Yaskawa INFORM job: test_long_tjr5.JBI

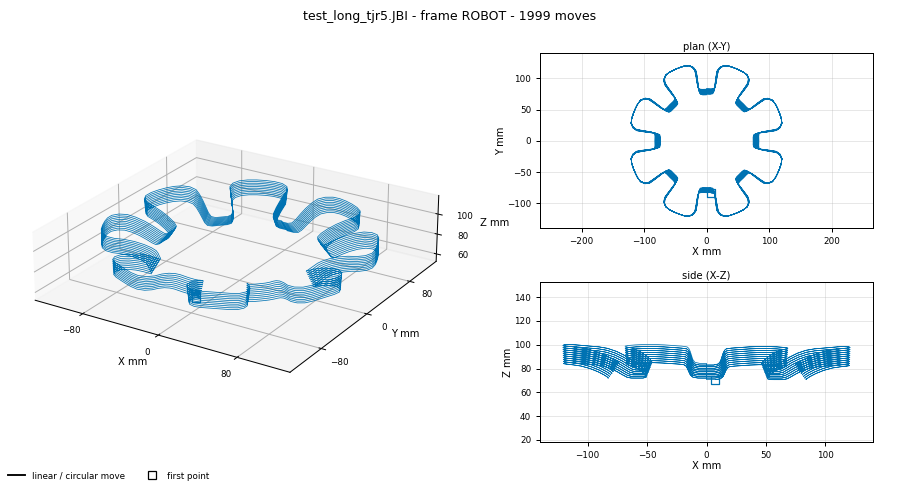
[picture p0: tool path of test_long_tjr5.JBI in frame ROBOT, 1999 of 2000 moves have a stored position in this frame; points joined in program order, loops and branches not executed]
version: 0
/JOB
//NAME test_long
//POS
///NPOS 48,0,0,2,0,0
///TOOL 1
///POSTYPE ROBOT
///RECTAN
///RCONF 1,0,0,0,0,0,0,0,0,0,0,0,0,0,0,0,0,0,0,0,0,0,0,0
C00000=3.480,-83.770,70.680,-0.0300,0.6200,0.7800
C00001=7.410,-83.590,70.710,0.0200,0.6100,0.7900
C00002=11.710,-84.200,71.430,0.2600,0.4000,0.8800
C00003=13.880,-86.990,73.260,0.0400,0.0100,1.0000
C00004=15.150,-91.900,75.810,-0.0600,-0.0100,1.0000
C00005=16.340,-98.510,78.470,-0.1100,-0.0200,0.9900
C00006=17.620,-105.970,80.520,-0.1300,-0.0300,0.9900
C00007=19.220,-112.910,81.540,-0.1300,-0.0600,0.9900
C00008=23.390,-117.950,82.080,-0.0500,-0.0700,1.0000
C00009=29.670,-120.290,82.520,-0.0000,-0.0400,1.0000
C00010=36.820,-119.400,82.970,0.0000,-0.0000,1.0000
C00011=44.160,-116.930,83.260,0.0000,-0.0000,1.0000
C00012=51.460,-113.910,83.260,0.0000,-0.0000,1.0000
C00013=58.390,-110.460,82.970,0.0000,-0.0000,1.0000
C00014=64.070,-106.040,82.520,0.0300,-0.0300,1.0000
C00015=66.860,-99.940,82.080,0.0800,-0.0200,1.0000
C00016=66.250,-93.430,81.540,0.1300,0.0500,0.9900
C00017=62.480,-87.390,80.520,0.1200,0.0700,0.9900
C00018=58.100,-81.210,78.470,0.0900,0.0600,0.9900
C00019=54.270,-75.700,75.810,0.0500,0.0300,1.0000
C00020=51.700,-71.330,73.260,-0.0400,-0.0200,1.0000
C00021=51.260,-67.810,71.430,-0.4700,0.1000,0.8800
C00022=53.870,-64.350,70.710,-0.4500,0.4200,0.7900
C00023=56.780,-61.700,70.680,-0.4200,0.4600,0.7800
C00024=59.280,-59.280,70.700,-0.4400,0.4400,0.7800
C00025=61.700,-56.780,70.680,-0.4600,0.4200,0.7800
C00026=64.350,-53.870,70.710,-0.4200,0.4500,0.7900
C00027=67.810,-51.260,71.430,-0.1000,0.4700,0.8800
C00028=71.330,-51.700,73.260,0.0200,0.0400,1.0000
C00029=75.700,-54.270,75.810,-0.0300,-0.0500,1.0000
C00030=81.210,-58.100,78.470,-0.0600,-0.0900,0.9900
C00031=87.390,-62.480,80.520,-0.0700,-0.1200,0.9900
C00032=93.430,-66.250,81.540,-0.0500,-0.1300,0.9900
C00033=99.940,-66.860,82.080,0.0200,-0.0800,1.0000
C00034=106.040,-64.070,82.520,0.0300,-0.0300,1.0000
C00035=110.460,-58.390,82.970,0.0000,-0.0000,1.0000
C00036=113.910,-51.460,83.260,0.0000,-0.0000,1.0000
C00037=116.930,-44.160,83.260,0.0000,-0.0000,1.0000
C00038=119.400,-36.820,82.970,0.0000,-0.0000,1.0000
C00039=120.290,-29.670,82.520,0.0400,0.0000,1.0000
C00040=117.950,-23.390,82.080,0.0700,0.0500,1.0000
C00041=112.910,-19.220,81.540,0.0600,0.1300,0.9900
C00042=105.970,-17.620,80.520,0.0300,0.1300,0.9900
C00043=98.510,-16.340,78.470,0.0200,0.1100,0.9900
C00044=91.900,-15.150,75.810,0.0100,0.0600,1.0000
C00045=86.990,-13.880,73.260,-0.0100,-0.0400,1.0000
C00046=84.200,-11.710,71.430,-0.4000,-0.2600,0.8800
C00047=83.590,-7.410,70.710,-0.6100,-0.0200,0.7900
C00048=83.770,-3.480,70.680,-0.6200,0.0300,0.7800
C00049=83.840,0.000,70.700,-0.6200,-0.0000,0.7800
C00050=83.770,3.480,70.680,-0.6200,-0.0300,0.7800
C00051=83.590,7.410,70.710,-0.6100,0.0200,0.7900
C00052=84.200,11.710,71.430,-0.4000,0.2600,0.8800
C00053=86.990,13.880,73.260,-0.0100,0.0400,1.0000
C00054=91.900,15.150,75.810,0.0100,-0.0600,1.0000
C00055=98.510,16.340,78.470,0.0200,-0.1100,0.9900
C00056=105.970,17.620,80.520,0.0300,-0.1300,0.9900
C00057=112.910,19.220,81.540,0.0600,-0.1300,0.9900
C00058=117.950,23.390,82.080,0.0700,-0.0500,1.0000
C00059=120.290,29.670,82.520,0.0400,-0.0000,1.0000
C00060=119.400,36.820,82.970,0.0000,0.0000,1.0000
C00061=116.930,44.160,83.260,0.0000,0.0000,1.0000
C00062=113.910,51.460,83.260,0.0000,0.0000,1.0000
C00063=110.460,58.390,82.970,0.0000,0.0000,1.0000
C00064=106.040,64.070,82.520,0.0300,0.0300,1.0000
C00065=99.940,66.860,82.080,0.0200,0.0800,1.0000
C00066=93.430,66.250,81.540,-0.0500,0.1300,0.9900
C00067=87.390,62.480,80.520,-0.0700,0.1200,0.9900
C00068=81.210,58.100,78.470,-0.0600,0.0900,0.9900
C00069=75.700,54.270,75.810,-0.0300,0.0500,1.0000
C00070=71.330,51.700,73.260,0.0200,-0.0400,1.0000
C00071=67.810,51.260,71.430,-0.1000,-0.4700,0.8800
C00072=64.350,53.870,70.710,-0.4200,-0.4500,0.7900
C00073=61.700,56.780,70.680,-0.4600,-0.4200,0.7800
C00074=59.280,59.280,70.700,-0.4400,-0.4400,0.7800
C00075=56.780,61.700,70.680,-0.4200,-0.4600,0.7800
C00076=53.870,64.350,70.710,-0.4500,-0.4200,0.7900
C00077=51.260,67.810,71.430,-0.4700,-0.1000,0.8800
C00078=51.700,71.330,73.260,-0.0400,0.0200,1.0000
C00079=54.270,75.700,75.810,0.0500,-0.0300,1.0000
C00080=58.100,81.210,78.470,0.0900,-0.0600,0.9900
C00081=62.480,87.390,80.520,0.1200,-0.0700,0.9900
C00082=66.250,93.430,81.540,0.1300,-0.0500,0.9900
C00083=66.860,99.940,82.080,0.0800,0.0200,1.0000
C00084=64.070,106.040,82.520,0.0300,0.0300,1.0000
C00085=58.390,110.460,82.970,0.0000,0.0000,1.0000
C00086=51.460,113.910,83.260,0.0000,0.0000,1.0000
C00087=44.160,116.930,83.260,0.0000,0.0000,1.0000
C00088=36.820,119.400,82.970,0.0000,0.0000,1.0000
C00089=29.670,120.290,82.520,-0.0000,0.0400,1.0000
C00090=23.390,117.950,82.080,-0.0500,0.0700,1.0000
C00091=19.220,112.910,81.540,-0.1300,0.0600,0.9900
C00092=17.620,105.970,80.520,-0.1300,0.0300,0.9900
C00093=16.340,98.510,78.470,-0.1100,0.0200,0.9900
C00094=15.150,91.900,75.810,-0.0600,0.0100,1.0000
C00095=13.880,86.990,73.260,0.0400,-0.0100,1.0000
C00096=11.710,84.200,71.430,0.2600,-0.4000,0.8800
C00097=7.410,83.590,70.710,0.0200,-0.6100,0.7900
C00098=3.480,83.770,70.680,-0.0300,-0.6200,0.7800
C00099=0.000,83.840,70.700,-0.0000,-0.6200,0.7800
C00100=0.000,82.790,72.040,-0.0000,-0.6200,0.7900
C00101=3.380,82.720,72.020,-0.0300,-0.6200,0.7900
C00102=7.250,82.550,72.050,0.0200,-0.6100,0.7900
C00103=11.510,83.190,72.790,0.2600,-0.3900,0.8800
C00104=13.630,86.090,74.680,0.0300,-0.0100,1.0000
C00105=14.880,91.140,77.300,-0.0600,0.0100,1.0000
C00106=16.050,97.940,80.040,-0.1100,0.0200,0.9900
C00107=17.310,105.610,82.150,-0.1300,0.0300,0.9900
C00108=18.890,112.730,83.200,-0.1300,0.0500,0.9900
C00109=23.080,117.910,83.750,-0.0500,0.0700,1.0000
C00110=29.430,120.330,84.200,-0.0100,0.0400,1.0000
C00111=36.670,119.450,84.660,0.0000,0.0000,1.0000
C00112=44.110,116.950,84.960,0.0000,0.0000,1.0000
C00113=51.510,113.890,84.960,0.0000,0.0000,1.0000
C00114=58.530,110.390,84.660,0.0000,0.0000,1.0000
C00115=64.280,105.900,84.200,0.0300,0.0300,1.0000
C00116=67.050,99.700,83.750,0.0800,0.0200,1.0000
C00117=66.360,93.070,83.200,0.1300,-0.0500,0.9900
C00118=62.440,86.920,82.150,0.1100,-0.0800,0.9900
C00119=57.910,80.600,80.040,0.0900,-0.0600,0.9900
C00120=53.930,74.970,77.300,0.0600,-0.0300,1.0000
C00121=51.230,70.510,74.680,-0.0300,0.0100,1.0000
C00122=50.690,66.970,72.790,-0.4600,-0.0900,0.8800
C00123=53.250,63.500,72.050,-0.4500,-0.4100,0.7900
C00124=56.100,60.890,72.020,-0.4200,-0.4600,0.7900
C00125=58.540,58.540,72.040,-0.4400,-0.4400,0.7900
C00126=60.890,56.100,72.020,-0.4600,-0.4200,0.7900
C00127=63.500,53.250,72.050,-0.4100,-0.4500,0.7900
C00128=66.970,50.690,72.790,-0.0900,-0.4600,0.8800
C00129=70.510,51.230,74.680,0.0100,-0.0300,1.0000
C00130=74.970,53.930,77.300,-0.0300,0.0600,1.0000
C00131=80.600,57.910,80.040,-0.0600,0.0900,0.9900
C00132=86.920,62.440,82.150,-0.0800,0.1100,0.9900
C00133=93.070,66.360,83.200,-0.0500,0.1300,0.9900
C00134=99.700,67.050,83.750,0.0200,0.0800,1.0000
C00135=105.900,64.280,84.200,0.0300,0.0300,1.0000
C00136=110.390,58.530,84.660,0.0000,0.0000,1.0000
C00137=113.890,51.510,84.960,0.0000,0.0000,1.0000
C00138=116.950,44.110,84.960,0.0000,0.0000,1.0000
C00139=119.450,36.670,84.660,0.0000,0.0000,1.0000
C00140=120.330,29.430,84.200,0.0400,-0.0100,1.0000
C00141=117.910,23.080,83.750,0.0700,-0.0500,1.0000
C00142=112.730,18.890,83.200,0.0500,-0.1300,0.9900
C00143=105.610,17.310,82.150,0.0300,-0.1300,0.9900
C00144=97.940,16.050,80.040,0.0200,-0.1100,0.9900
C00145=91.140,14.880,77.300,0.0100,-0.0600,1.0000
C00146=86.090,13.630,74.680,-0.0100,0.0300,1.0000
C00147=83.190,11.510,72.790,-0.3900,0.2600,0.8800
C00148=82.550,7.250,72.050,-0.6100,0.0200,0.7900
C00149=82.720,3.380,72.020,-0.6200,-0.0300,0.7900
C00150=82.790,0.000,72.040,-0.6200,-0.0000,0.7900
C00151=82.720,-3.380,72.020,-0.6200,0.0300,0.7900
C00152=82.550,-7.250,72.050,-0.6100,-0.0200,0.7900
C00153=83.190,-11.510,72.790,-0.3900,-0.2600,0.8800
C00154=86.090,-13.630,74.680,-0.0100,-0.0300,1.0000
C00155=91.140,-14.880,77.300,0.0100,0.0600,1.0000
C00156=97.940,-16.050,80.040,0.0200,0.1100,0.9900
C00157=105.610,-17.310,82.150,0.0300,0.1300,0.9900
C00158=112.730,-18.890,83.200,0.0500,0.1300,0.9900
C00159=117.910,-23.080,83.750,0.0700,0.0500,1.0000
C00160=120.330,-29.430,84.200,0.0400,0.0100,1.0000
C00161=119.450,-36.670,84.660,0.0000,-0.0000,1.0000
C00162=116.950,-44.110,84.960,0.0000,-0.0000,1.0000
C00163=113.890,-51.510,84.960,0.0000,-0.0000,1.0000
C00164=110.390,-58.530,84.660,0.0000,-0.0000,1.0000
C00165=105.900,-64.280,84.200,0.0300,-0.0300,1.0000
C00166=99.700,-67.050,83.750,0.0200,-0.0800,1.0000
C00167=93.070,-66.360,83.200,-0.0500,-0.1300,0.9900
C00168=86.920,-62.440,82.150,-0.0800,-0.1100,0.9900
C00169=80.600,-57.910,80.040,-0.0600,-0.0900,0.9900
C00170=74.970,-53.930,77.300,-0.0300,-0.0600,1.0000
C00171=70.510,-51.230,74.680,0.0100,0.0300,1.0000
C00172=66.970,-50.690,72.790,-0.0900,0.4600,0.8800
C00173=63.500,-53.250,72.050,-0.4100,0.4500,0.7900
C00174=60.890,-56.100,72.020,-0.4600,0.4200,0.7900
C00175=58.540,-58.540,72.040,-0.4400,0.4400,0.7900
C00176=56.100,-60.890,72.020,-0.4200,0.4600,0.7900
C00177=53.250,-63.500,72.050,-0.4500,0.4100,0.7900
C00178=50.690,-66.970,72.790,-0.4600,0.0900,0.8800
C00179=51.230,-70.510,74.680,-0.0300,-0.0100,1.0000
C00180=53.930,-74.970,77.300,0.0600,0.0300,1.0000
C00181=57.910,-80.600,80.040,0.0900,0.0600,0.9900
C00182=62.440,-86.920,82.150,0.1100,0.0800,0.9900
C00183=66.360,-93.070,83.200,0.1300,0.0500,0.9900
C00184=67.050,-99.700,83.750,0.0800,-0.0200,1.0000
C00185=64.280,-105.900,84.200,0.0300,-0.0300,1.0000
C00186=58.530,-110.390,84.660,0.0000,-0.0000,1.0000
C00187=51.510,-113.890,84.960,0.0000,-0.0000,1.0000
C00188=44.110,-116.950,84.960,0.0000,-0.0000,1.0000
C00189=36.670,-119.450,84.660,0.0000,-0.0000,1.0000
C00190=29.430,-120.330,84.200,-0.0100,-0.0400,1.0000
C00191=23.080,-117.910,83.750,-0.0500,-0.0700,1.0000
C00192=18.890,-112.730,83.200,-0.1300,-0.0500,0.9900
C00193=17.310,-105.610,82.150,-0.1300,-0.0300,0.9900
C00194=16.050,-97.940,80.040,-0.1100,-0.0200,0.9900
C00195=14.880,-91.140,77.300,-0.0600,-0.0100,1.0000
C00196=13.630,-86.090,74.680,0.0300,0.0100,1.0000
C00197=11.510,-83.190,72.790,0.2600,0.3900,0.8800
C00198=7.250,-82.550,72.050,0.0200,0.6100,0.7900
C00199=3.380,-82.720,72.020,-0.0300,0.6200,0.7900
C00200=0.000,-82.790,72.040,-0.0000,0.6200,0.7900
C00201=0.000,-82.790,72.040,-0.0000,0.6200,0.7900
C00202=-3.380,-82.720,72.020,0.0300,0.6200,0.7900
C00203=-7.250,-82.550,72.050,-0.0200,0.6100,0.7900
C00204=-11.510,-83.190,72.790,-0.2600,0.3900,0.8800
C00205=-13.630,-86.090,74.680,-0.0300,0.0100,1.0000
C00206=-14.880,-91.140,77.300,0.0600,-0.0100,1.0000
C00207=-16.050,-97.940,80.040,0.1100,-0.0200,0.9900
C00208=-17.310,-105.610,82.150,0.1300,-0.0300,0.9900
C00209=-18.890,-112.730,83.200,0.1300,-0.0500,0.9900
C00210=-23.080,-117.910,83.750,0.0500,-0.0700,1.0000
C00211=-29.430,-120.330,84.200,0.0100,-0.0400,1.0000
C00212=-36.670,-119.450,84.660,-0.0000,-0.0000,1.0000
C00213=-44.110,-116.950,84.960,-0.0000,-0.0000,1.0000
C00214=-51.510,-113.890,84.960,-0.0000,-0.0000,1.0000
C00215=-58.530,-110.390,84.660,-0.0000,-0.0000,1.0000
C00216=-64.280,-105.900,84.200,-0.0300,-0.0300,1.0000
C00217=-67.050,-99.700,83.750,-0.0800,-0.0200,1.0000
C00218=-66.360,-93.070,83.200,-0.1300,0.0500,0.9900
C00219=-62.440,-86.920,82.150,-0.1100,0.0800,0.9900
C00220=-57.910,-80.600,80.040,-0.0900,0.0600,0.9900
C00221=-53.930,-74.970,77.300,-0.0600,0.0300,1.0000
C00222=-51.230,-70.510,74.680,0.0300,-0.0100,1.0000
C00223=-50.690,-66.970,72.790,0.4600,0.0900,0.8800
C00224=-53.250,-63.500,72.050,0.4500,0.4100,0.7900
C00225=-56.100,-60.890,72.020,0.4200,0.4600,0.7900
C00226=-58.540,-58.540,72.040,0.4400,0.4400,0.7900
C00227=-60.890,-56.100,72.020,0.4600,0.4200,0.7900
C00228=-63.500,-53.250,72.050,0.4100,0.4500,0.7900
C00229=-66.970,-50.690,72.790,0.0900,0.4600,0.8800
C00230=-70.510,-51.230,74.680,-0.0100,0.0300,1.0000
C00231=-74.970,-53.930,77.300,0.0300,-0.0600,1.0000
C00232=-80.600,-57.910,80.040,0.0600,-0.0900,0.9900
C00233=-86.920,-62.440,82.150,0.0800,-0.1100,0.9900
C00234=-93.070,-66.360,83.200,0.0500,-0.1300,0.9900
C00235=-99.700,-67.050,83.750,-0.0200,-0.0800,1.0000
C00236=-105.900,-64.280,84.200,-0.0300,-0.0300,1.0000
C00237=-110.390,-58.530,84.660,-0.0000,-0.0000,1.0000
C00238=-113.890,-51.510,84.960,-0.0000,-0.0000,1.0000
C00239=-116.950,-44.110,84.960,-0.0000,-0.0000,1.0000
C00240=-119.450,-36.670,84.660,-0.0000,-0.0000,1.0000
C00241=-120.330,-29.430,84.200,-0.0400,0.0100,1.0000
C00242=-117.910,-23.080,83.750,-0.0700,0.0500,1.0000
C00243=-112.730,-18.890,83.200,-0.0500,0.1300,0.9900
C00244=-105.610,-17.310,82.150,-0.0300,0.1300,0.9900
C00245=-97.940,-16.050,80.040,-0.0200,0.1100,0.9900
C00246=-91.140,-14.880,77.300,-0.0100,0.0600,1.0000
C00247=-86.090,-13.630,74.680,0.0100,-0.0300,1.0000
C00248=-83.190,-11.510,72.790,0.3900,-0.2600,0.8800
C00249=-82.550,-7.250,72.050,0.6100,-0.0200,0.7900
C00250=-82.720,-3.380,72.020,0.6200,0.0300,0.7900
C00251=-82.790,0.000,72.040,0.6200,0.0000,0.7900
C00252=-82.720,3.380,72.020,0.6200,-0.0300,0.7900
C00253=-82.550,7.250,72.050,0.6100,0.0200,0.7900
C00254=-83.190,11.510,72.790,0.3900,0.2600,0.8800
C00255=-86.090,13.630,74.680,0.0100,0.0300,1.0000
C00256=-91.140,14.880,77.300,-0.0100,-0.0600,1.0000
C00257=-97.940,16.050,80.040,-0.0200,-0.1100,0.9900
C00258=-105.610,17.310,82.150,-0.0300,-0.1300,0.9900
C00259=-112.730,18.890,83.200,-0.0500,-0.1300,0.9900
C00260=-117.910,23.080,83.750,-0.0700,-0.0500,1.0000
C00261=-120.330,29.430,84.200,-0.0400,-0.0100,1.0000
C00262=-119.450,36.670,84.660,-0.0000,0.0000,1.0000
C00263=-116.950,44.110,84.960,-0.0000,0.0000,1.0000
C00264=-113.890,51.510,84.960,-0.0000,0.0000,1.0000
C00265=-110.390,58.530,84.660,-0.0000,0.0000,1.0000
C00266=-105.900,64.280,84.200,-0.0300,0.0300,1.0000
C00267=-99.700,67.050,83.750,-0.0200,0.0800,1.0000
C00268=-93.070,66.360,83.200,0.0500,0.1300,0.9900
C00269=-86.920,62.440,82.150,0.0800,0.1100,0.9900
C00270=-80.600,57.910,80.040,0.0600,0.0900,0.9900
C00271=-74.970,53.930,77.300,0.0300,0.0600,1.0000
C00272=-70.510,51.230,74.680,-0.0100,-0.0300,1.0000
C00273=-66.970,50.690,72.790,0.0900,-0.4600,0.8800
C00274=-63.500,53.250,72.050,0.4100,-0.4500,0.7900
C00275=-60.890,56.100,72.020,0.4600,-0.4200,0.7900
C00276=-58.540,58.540,72.040,0.4400,-0.4400,0.7900
C00277=-56.100,60.890,72.020,0.4200,-0.4600,0.7900
C00278=-53.250,63.500,72.050,0.4500,-0.4100,0.7900
C00279=-50.690,66.970,72.790,0.4600,-0.0900,0.8800
C00280=-51.230,70.510,74.680,0.0300,0.0100,1.0000
C00281=-53.930,74.970,77.300,-0.0600,-0.0300,1.0000
C00282=-57.910,80.600,80.040,-0.0900,-0.0600,0.9900
C00283=-62.440,86.920,82.150,-0.1100,-0.0800,0.9900
C00284=-66.360,93.070,83.200,-0.1300,-0.0500,0.9900
C00285=-67.050,99.700,83.750,-0.0800,0.0200,1.0000
C00286=-64.280,105.900,84.200,-0.0300,0.0300,1.0000
C00287=-58.530,110.390,84.660,-0.0000,0.0000,1.0000
C00288=-51.510,113.890,84.960,-0.0000,0.0000,1.0000
C00289=-44.110,116.950,84.960,-0.0000,0.0000,1.0000
C00290=-36.670,119.450,84.660,-0.0000,0.0000,1.0000
C00291=-29.430,120.330,84.200,0.0100,0.0400,1.0000
C00292=-23.080,117.910,83.750,0.0500,0.0700,1.0000
C00293=-18.890,112.730,83.200,0.1300,0.0500,0.9900
C00294=-17.310,105.610,82.150,0.1300,0.0300,0.9900
C00295=-16.050,97.940,80.040,0.1100,0.0200,0.9900
C00296=-14.880,91.140,77.300,0.0600,0.0100,1.0000
C00297=-13.630,86.090,74.680,-0.0300,-0.0100,1.0000
C00298=-11.510,83.190,72.790,-0.2600,-0.3900,0.8800
C00299=-7.250,82.550,72.050,-0.0200,-0.6100,0.7900
C00300=-3.380,82.720,72.020,0.0300,-0.6200,0.7900
C00301=0.000,82.790,72.040,-0.0000,-0.6200,0.7900
C00302=0.000,81.740,73.380,-0.0000,-0.6100,0.7900
C00303=-3.290,81.680,73.350,0.0300,-0.6100,0.7900
C00304=-7.090,81.520,73.390,-0.0300,-0.6000,0.8000
C00305=-11.310,82.200,74.160,-0.2600,-0.3800,0.8900
C00306=-13.400,85.190,76.100,-0.0200,-0.0100,1.0000
C00307=-14.610,90.400,78.810,0.0700,0.0100,1.0000
C00308=-15.760,97.380,81.620,0.1100,0.0200,0.9900
C00309=-17.010,105.250,83.790,0.1300,0.0300,0.9900
C00310=-18.570,112.560,84.860,0.1300,0.0500,0.9900
C00311=-22.780,117.880,85.430,0.0500,0.0700,1.0000
C00312=-29.200,120.370,85.890,0.0100,0.0400,1.0000
C00313=-36.520,119.490,86.350,-0.0000,0.0000,1.0000
C00314=-44.060,116.970,86.660,-0.0000,0.0000,1.0000
C00315=-51.560,113.870,86.660,-0.0000,0.0000,1.0000
C00316=-58.670,110.320,86.350,-0.0000,0.0000,1.0000
C00317=-64.470,105.760,85.890,-0.0300,0.0300,1.0000
C00318=-67.240,99.460,85.430,-0.0800,0.0100,1.0000
C00319=-66.460,92.720,84.860,-0.1300,-0.0500,0.9900
C00320=-62.400,86.450,83.790,-0.1100,-0.0700,0.9900
C00321=-57.710,80.010,81.620,-0.0900,-0.0600,0.9900
C00322=-53.590,74.250,78.810,-0.0600,-0.0400,1.0000
C00323=-50.760,69.710,76.100,0.0200,0.0100,1.0000
C00324=-50.120,66.120,74.160,0.4500,-0.0800,0.8900
C00325=-52.630,62.650,73.390,0.4500,-0.4100,0.8000
C00326=-55.430,60.080,73.350,0.4100,-0.4500,0.7900
C00327=-57.800,57.800,73.380,0.4300,-0.4300,0.7900
C00328=-60.080,55.430,73.350,0.4500,-0.4100,0.7900
C00329=-62.650,52.630,73.390,0.4100,-0.4500,0.8000
C00330=-66.120,50.120,74.160,0.0800,-0.4500,0.8900
C00331=-69.710,50.760,76.100,-0.0100,-0.0200,1.0000
C00332=-74.250,53.590,78.810,0.0400,0.0600,1.0000
C00333=-80.010,57.710,81.620,0.0600,0.0900,0.9900
C00334=-86.450,62.400,83.790,0.0700,0.1100,0.9900
C00335=-92.720,66.460,84.860,0.0500,0.1300,0.9900
C00336=-99.460,67.240,85.430,-0.0100,0.0800,1.0000
C00337=-105.760,64.470,85.890,-0.0300,0.0300,1.0000
C00338=-110.320,58.670,86.350,-0.0000,0.0000,1.0000
C00339=-113.870,51.560,86.660,-0.0000,0.0000,1.0000
C00340=-116.970,44.060,86.660,-0.0000,0.0000,1.0000
C00341=-119.490,36.520,86.350,-0.0000,0.0000,1.0000
C00342=-120.370,29.200,85.890,-0.0400,-0.0100,1.0000
C00343=-117.880,22.780,85.430,-0.0700,-0.0500,1.0000
C00344=-112.560,18.570,84.860,-0.0500,-0.1300,0.9900
C00345=-105.250,17.010,83.790,-0.0300,-0.1300,0.9900
C00346=-97.380,15.760,81.620,-0.0200,-0.1100,0.9900
C00347=-90.400,14.610,78.810,-0.0100,-0.0700,1.0000
C00348=-85.190,13.400,76.100,0.0100,0.0200,1.0000
C00349=-82.200,11.310,74.160,0.3800,0.2600,0.8900
C00350=-81.520,7.090,73.390,0.6000,0.0300,0.8000
C00351=-81.680,3.290,73.350,0.6100,-0.0300,0.7900
C00352=-81.740,0.000,73.380,0.6100,0.0000,0.7900
C00353=-81.680,-3.290,73.350,0.6100,0.0300,0.7900
C00354=-81.520,-7.090,73.390,0.6000,-0.0300,0.8000
C00355=-82.200,-11.310,74.160,0.3800,-0.2600,0.8900
C00356=-85.190,-13.400,76.100,0.0100,-0.0200,1.0000
C00357=-90.400,-14.610,78.810,-0.0100,0.0700,1.0000
C00358=-97.380,-15.760,81.620,-0.0200,0.1100,0.9900
C00359=-105.250,-17.010,83.790,-0.0300,0.1300,0.9900
C00360=-112.560,-18.570,84.860,-0.0500,0.1300,0.9900
C00361=-117.880,-22.780,85.430,-0.0700,0.0500,1.0000
C00362=-120.370,-29.200,85.890,-0.0400,0.0100,1.0000
C00363=-119.490,-36.520,86.350,-0.0000,-0.0000,1.0000
C00364=-116.970,-44.060,86.660,-0.0000,-0.0000,1.0000
C00365=-113.870,-51.560,86.660,-0.0000,-0.0000,1.0000
C00366=-110.320,-58.670,86.350,-0.0000,-0.0000,1.0000
C00367=-105.760,-64.470,85.890,-0.0300,-0.0300,1.0000
C00368=-99.460,-67.240,85.430,-0.0100,-0.0800,1.0000
C00369=-92.720,-66.460,84.860,0.0500,-0.1300,0.9900
C00370=-86.450,-62.400,83.790,0.0700,-0.1100,0.9900
C00371=-80.010,-57.710,81.620,0.0600,-0.0900,0.9900
C00372=-74.250,-53.590,78.810,0.0400,-0.0600,1.0000
C00373=-69.710,-50.760,76.100,-0.0100,0.0200,1.0000
C00374=-66.120,-50.120,74.160,0.0800,0.4500,0.8900
C00375=-62.650,-52.630,73.390,0.4100,0.4500,0.8000
C00376=-60.080,-55.430,73.350,0.4500,0.4100,0.7900
C00377=-57.800,-57.800,73.380,0.4300,0.4300,0.7900
C00378=-55.430,-60.080,73.350,0.4100,0.4500,0.7900
C00379=-52.630,-62.650,73.390,0.4500,0.4100,0.8000
C00380=-50.120,-66.120,74.160,0.4500,0.0800,0.8900
C00381=-50.760,-69.710,76.100,0.0200,-0.0100,1.0000
C00382=-53.590,-74.250,78.810,-0.0600,0.0400,1.0000
C00383=-57.710,-80.010,81.620,-0.0900,0.0600,0.9900
C00384=-62.400,-86.450,83.790,-0.1100,0.0700,0.9900
C00385=-66.460,-92.720,84.860,-0.1300,0.0500,0.9900
C00386=-67.240,-99.460,85.430,-0.0800,-0.0100,1.0000
C00387=-64.470,-105.760,85.890,-0.0300,-0.0300,1.0000
C00388=-58.670,-110.320,86.350,-0.0000,-0.0000,1.0000
C00389=-51.560,-113.870,86.660,-0.0000,-0.0000,1.0000
C00390=-44.060,-116.970,86.660,-0.0000,-0.0000,1.0000
C00391=-36.520,-119.490,86.350,-0.0000,-0.0000,1.0000
C00392=-29.200,-120.370,85.890,0.0100,-0.0400,1.0000
C00393=-22.780,-117.880,85.430,0.0500,-0.0700,1.0000
C00394=-18.570,-112.560,84.860,0.1300,-0.0500,0.9900
C00395=-17.010,-105.250,83.790,0.1300,-0.0300,0.9900
C00396=-15.760,-97.380,81.620,0.1100,-0.0200,0.9900
C00397=-14.610,-90.400,78.810,0.0700,-0.0100,1.0000
C00398=-13.400,-85.190,76.100,-0.0200,0.0100,1.0000
C00399=-11.310,-82.200,74.160,-0.2600,0.3800,0.8900
C00400=-7.090,-81.520,73.390,-0.0300,0.6000,0.8000
C00401=-3.290,-81.680,73.350,0.0300,0.6100,0.7900
C00402=0.000,-81.740,73.380,-0.0000,0.6100,0.7900
C00403=0.000,-81.740,73.380,-0.0000,0.6100,0.7900
C00404=3.290,-81.680,73.350,-0.0300,0.6100,0.7900
C00405=7.090,-81.520,73.390,0.0300,0.6000,0.8000
C00406=11.310,-82.200,74.160,0.2600,0.3800,0.8900
C00407=13.400,-85.190,76.100,0.0200,0.0100,1.0000
C00408=14.610,-90.400,78.810,-0.0700,-0.0100,1.0000
C00409=15.760,-97.380,81.620,-0.1100,-0.0200,0.9900
C00410=17.010,-105.250,83.790,-0.1300,-0.0300,0.9900
C00411=18.570,-112.560,84.860,-0.1300,-0.0500,0.9900
C00412=22.780,-117.880,85.430,-0.0500,-0.0700,1.0000
C00413=29.200,-120.370,85.890,-0.0100,-0.0400,1.0000
C00414=36.520,-119.490,86.350,0.0000,-0.0000,1.0000
C00415=44.060,-116.970,86.660,0.0000,-0.0000,1.0000
C00416=51.560,-113.870,86.660,0.0000,-0.0000,1.0000
C00417=58.670,-110.320,86.350,0.0000,-0.0000,1.0000
C00418=64.470,-105.760,85.890,0.0300,-0.0300,1.0000
C00419=67.240,-99.460,85.430,0.0800,-0.0100,1.0000
C00420=66.460,-92.720,84.860,0.1300,0.0500,0.9900
C00421=62.400,-86.450,83.790,0.1100,0.0700,0.9900
C00422=57.710,-80.010,81.620,0.0900,0.0600,0.9900
C00423=53.590,-74.250,78.810,0.0600,0.0400,1.0000
C00424=50.760,-69.710,76.100,-0.0200,-0.0100,1.0000
C00425=50.120,-66.120,74.160,-0.4500,0.0800,0.8900
C00426=52.630,-62.650,73.390,-0.4500,0.4100,0.8000
C00427=55.430,-60.080,73.350,-0.4100,0.4500,0.7900
C00428=57.800,-57.800,73.380,-0.4300,0.4300,0.7900
C00429=60.080,-55.430,73.350,-0.4500,0.4100,0.7900
C00430=62.650,-52.630,73.390,-0.4100,0.4500,0.8000
C00431=66.120,-50.120,74.160,-0.0800,0.4500,0.8900
C00432=69.710,-50.760,76.100,0.0100,0.0200,1.0000
C00433=74.250,-53.590,78.810,-0.0400,-0.0600,1.0000
C00434=80.010,-57.710,81.620,-0.0600,-0.0900,0.9900
C00435=86.450,-62.400,83.790,-0.0700,-0.1100,0.9900
C00436=92.720,-66.460,84.860,-0.0500,-0.1300,0.9900
C00437=99.460,-67.240,85.430,0.0100,-0.0800,1.0000
C00438=105.760,-64.470,85.890,0.0300,-0.0300,1.0000
C00439=110.320,-58.670,86.350,0.0000,-0.0000,1.0000
C00440=113.870,-51.560,86.660,0.0000,-0.0000,1.0000
C00441=116.970,-44.060,86.660,0.0000,-0.0000,1.0000
C00442=119.490,-36.520,86.350,0.0000,-0.0000,1.0000
C00443=120.370,-29.200,85.890,0.0400,0.0100,1.0000
C00444=117.880,-22.780,85.430,0.0700,0.0500,1.0000
C00445=112.560,-18.570,84.860,0.0500,0.1300,0.9900
C00446=105.250,-17.010,83.790,0.0300,0.1300,0.9900
C00447=97.380,-15.760,81.620,0.0200,0.1100,0.9900
C00448=90.400,-14.610,78.810,0.0100,0.0700,1.0000
C00449=85.190,-13.400,76.100,-0.0100,-0.0200,1.0000
C00450=82.200,-11.310,74.160,-0.3800,-0.2600,0.8900
C00451=81.520,-7.090,73.390,-0.6000,-0.0300,0.8000
C00452=81.680,-3.290,73.350,-0.6100,0.0300,0.7900
C00453=81.740,0.000,73.380,-0.6100,-0.0000,0.7900
C00454=81.680,3.290,73.350,-0.6100,-0.0300,0.7900
C00455=81.520,7.090,73.390,-0.6000,0.0300,0.8000
C00456=82.200,11.310,74.160,-0.3800,0.2600,0.8900
C00457=85.190,13.400,76.100,-0.0100,0.0200,1.0000
C00458=90.400,14.610,78.810,0.0100,-0.0700,1.0000
C00459=97.380,15.760,81.620,0.0200,-0.1100,0.9900
C00460=105.250,17.010,83.790,0.0300,-0.1300,0.9900
C00461=112.560,18.570,84.860,0.0500,-0.1300,0.9900
C00462=117.880,22.780,85.430,0.0700,-0.0500,1.0000
C00463=120.370,29.200,85.890,0.0400,-0.0100,1.0000
C00464=119.490,36.520,86.350,0.0000,0.0000,1.0000
C00465=116.970,44.060,86.660,0.0000,0.0000,1.0000
C00466=113.870,51.560,86.660,0.0000,0.0000,1.0000
C00467=110.320,58.670,86.350,0.0000,0.0000,1.0000
C00468=105.760,64.470,85.890,0.0300,0.0300,1.0000
C00469=99.460,67.240,85.430,0.0100,0.0800,1.0000
C00470=92.720,66.460,84.860,-0.0500,0.1300,0.9900
C00471=86.450,62.400,83.790,-0.0700,0.1100,0.9900
C00472=80.010,57.710,81.620,-0.0600,0.0900,0.9900
C00473=74.250,53.590,78.810,-0.0400,0.0600,1.0000
C00474=69.710,50.760,76.100,0.0100,-0.0200,1.0000
C00475=66.120,50.120,74.160,-0.0800,-0.4500,0.8900
C00476=62.650,52.630,73.390,-0.4100,-0.4500,0.8000
C00477=60.080,55.430,73.350,-0.4500,-0.4100,0.7900
C00478=57.800,57.800,73.380,-0.4300,-0.4300,0.7900
C00479=55.430,60.080,73.350,-0.4100,-0.4500,0.7900
C00480=52.630,62.650,73.390,-0.4500,-0.4100,0.8000
C00481=50.120,66.120,74.160,-0.4500,-0.0800,0.8900
C00482=50.760,69.710,76.100,-0.0200,0.0100,1.0000
C00483=53.590,74.250,78.810,0.0600,-0.0400,1.0000
C00484=57.710,80.010,81.620,0.0900,-0.0600,0.9900
C00485=62.400,86.450,83.790,0.1100,-0.0700,0.9900
C00486=66.460,92.720,84.860,0.1300,-0.0500,0.9900
C00487=67.240,99.460,85.430,0.0800,0.0100,1.0000
C00488=64.470,105.760,85.890,0.0300,0.0300,1.0000
C00489=58.670,110.320,86.350,0.0000,0.0000,1.0000
C00490=51.560,113.870,86.660,0.0000,0.0000,1.0000
C00491=44.060,116.970,86.660,0.0000,0.0000,1.0000
C00492=36.520,119.490,86.350,0.0000,0.0000,1.0000
C00493=29.200,120.370,85.890,-0.0100,0.0400,1.0000
C00494=22.780,117.880,85.430,-0.0500,0.0700,1.0000
C00495=18.570,112.560,84.860,-0.1300,0.0500,0.9900
C00496=17.010,105.250,83.790,-0.1300,0.0300,0.9900
C00497=15.760,97.380,81.620,-0.1100,0.0200,0.9900
C00498=14.610,90.400,78.810,-0.0700,0.0100,1.0000
C00499=13.400,85.190,76.100,0.0200,-0.0100,1.0000
C00500=11.310,82.200,74.160,0.2600,-0.3800,0.8900
C00501=7.090,81.520,73.390,0.0300,-0.6000,0.8000
C00502=3.290,81.680,73.350,-0.0300,-0.6100,0.7900
C00503=0.000,81.740,73.380,-0.0000,-0.6100,0.7900
C00504=0.000,80.700,74.720,-0.0000,-0.6100,0.7900
C00505=3.190,80.650,74.700,-0.0300,-0.6100,0.7900
C00506=6.930,80.490,74.730,0.0300,-0.6000,0.8000
C00507=11.120,81.210,75.530,0.2600,-0.3600,0.8900
C00508=13.160,84.300,77.530,0.0100,-0.0000,1.0000
C00509=14.350,89.660,80.320,-0.0700,0.0100,1.0000
C00510=15.480,96.840,83.210,-0.1100,0.0200,0.9900
C00511=16.720,104.900,85.430,-0.1300,0.0200,0.9900
C00512=18.250,112.380,86.520,-0.1200,0.0500,0.9900
C00513=22.490,117.840,87.100,-0.0500,0.0700,1.0000
C00514=28.970,120.420,87.570,-0.0100,0.0400,1.0000
C00515=36.370,119.540,88.050,0.0000,0.0000,1.0000
C00516=44.010,116.990,88.360,0.0000,0.0000,1.0000
C00517=51.610,113.840,88.360,0.0000,0.0000,1.0000
C00518=58.810,110.250,88.050,0.0000,0.0000,1.0000
C00519=64.670,105.630,87.570,0.0300,0.0300,1.0000
C00520=67.420,99.230,87.100,0.0800,0.0100,1.0000
C00521=66.560,92.380,86.520,0.1200,-0.0500,0.9900
C00522=62.360,86.000,85.430,0.1100,-0.0700,0.9900
C00523=57.530,79.420,83.210,0.0900,-0.0600,0.9900
C00524=53.250,73.540,80.320,0.0600,-0.0400,1.0000
C00525=50.300,68.910,77.530,-0.0100,0.0100,1.0000
C00526=49.560,65.290,75.530,-0.4400,-0.0700,0.8900
C00527=52.020,61.810,74.730,-0.4500,-0.4000,0.8000
C00528=54.770,59.280,74.700,-0.4100,-0.4500,0.7900
C00529=57.070,57.070,74.720,-0.4300,-0.4300,0.7900
C00530=59.280,54.770,74.700,-0.4500,-0.4100,0.7900
C00531=61.810,52.020,74.730,-0.4000,-0.4500,0.8000
C00532=65.290,49.560,75.530,-0.0700,-0.4400,0.8900
C00533=68.910,50.300,77.530,0.0100,-0.0100,1.0000
C00534=73.540,53.250,80.320,-0.0400,0.0600,1.0000
C00535=79.420,57.530,83.210,-0.0600,0.0900,0.9900
C00536=86.000,62.360,85.430,-0.0700,0.1100,0.9900
C00537=92.380,66.560,86.520,-0.0500,0.1200,0.9900
C00538=99.230,67.420,87.100,0.0100,0.0800,1.0000
C00539=105.630,64.670,87.570,0.0300,0.0300,1.0000
C00540=110.250,58.810,88.050,0.0000,0.0000,1.0000
C00541=113.840,51.610,88.360,0.0000,0.0000,1.0000
C00542=116.990,44.010,88.360,0.0000,0.0000,1.0000
C00543=119.540,36.370,88.050,0.0000,0.0000,1.0000
C00544=120.420,28.970,87.570,0.0400,-0.0100,1.0000
C00545=117.840,22.490,87.100,0.0700,-0.0500,1.0000
C00546=112.380,18.250,86.520,0.0500,-0.1200,0.9900
C00547=104.900,16.720,85.430,0.0200,-0.1300,0.9900
C00548=96.840,15.480,83.210,0.0200,-0.1100,0.9900
C00549=89.660,14.350,80.320,0.0100,-0.0700,1.0000
C00550=84.300,13.160,77.530,-0.0000,0.0100,1.0000
C00551=81.210,11.120,75.530,-0.3600,0.2600,0.8900
C00552=80.490,6.930,74.730,-0.6000,0.0300,0.8000
C00553=80.650,3.190,74.700,-0.6100,-0.0300,0.7900
C00554=80.700,0.000,74.720,-0.6100,-0.0000,0.7900
C00555=80.650,-3.190,74.700,-0.6100,0.0300,0.7900
C00556=80.490,-6.930,74.730,-0.6000,-0.0300,0.8000
C00557=81.210,-11.120,75.530,-0.3600,-0.2600,0.8900
C00558=84.300,-13.160,77.530,-0.0000,-0.0100,1.0000
C00559=89.660,-14.350,80.320,0.0100,0.0700,1.0000
C00560=96.840,-15.480,83.210,0.0200,0.1100,0.9900
C00561=104.900,-16.720,85.430,0.0200,0.1300,0.9900
C00562=112.380,-18.250,86.520,0.0500,0.1200,0.9900
C00563=117.840,-22.490,87.100,0.0700,0.0500,1.0000
C00564=120.420,-28.970,87.570,0.0400,0.0100,1.0000
C00565=119.540,-36.370,88.050,0.0000,-0.0000,1.0000
C00566=116.990,-44.010,88.360,0.0000,-0.0000,1.0000
C00567=113.840,-51.610,88.360,0.0000,-0.0000,1.0000
C00568=110.250,-58.810,88.050,0.0000,-0.0000,1.0000
C00569=105.630,-64.670,87.570,0.0300,-0.0300,1.0000
C00570=99.230,-67.420,87.100,0.0100,-0.0800,1.0000
C00571=92.380,-66.560,86.520,-0.0500,-0.1200,0.9900
C00572=86.000,-62.360,85.430,-0.0700,-0.1100,0.9900
C00573=79.420,-57.530,83.210,-0.0600,-0.0900,0.9900
C00574=73.540,-53.250,80.320,-0.0400,-0.0600,1.0000
C00575=68.910,-50.300,77.530,0.0100,0.0100,1.0000
C00576=65.290,-49.560,75.530,-0.0700,0.4400,0.8900
C00577=61.810,-52.020,74.730,-0.4000,0.4500,0.8000
C00578=59.280,-54.770,74.700,-0.4500,0.4100,0.7900
C00579=57.070,-57.070,74.720,-0.4300,0.4300,0.7900
C00580=54.770,-59.280,74.700,-0.4100,0.4500,0.7900
C00581=52.020,-61.810,74.730,-0.4500,0.4000,0.8000
C00582=49.560,-65.290,75.530,-0.4400,0.0700,0.8900
C00583=50.300,-68.910,77.530,-0.0100,-0.0100,1.0000
C00584=53.250,-73.540,80.320,0.0600,0.0400,1.0000
C00585=57.530,-79.420,83.210,0.0900,0.0600,0.9900
C00586=62.360,-86.000,85.430,0.1100,0.0700,0.9900
C00587=66.560,-92.380,86.520,0.1200,0.0500,0.9900
C00588=67.420,-99.230,87.100,0.0800,-0.0100,1.0000
C00589=64.670,-105.630,87.570,0.0300,-0.0300,1.0000
C00590=58.810,-110.250,88.050,0.0000,-0.0000,1.0000
C00591=51.610,-113.840,88.360,0.0000,-0.0000,1.0000
C00592=44.010,-116.990,88.360,0.0000,-0.0000,1.0000
C00593=36.370,-119.540,88.050,0.0000,-0.0000,1.0000
C00594=28.970,-120.420,87.570,-0.0100,-0.0400,1.0000
C00595=22.490,-117.840,87.100,-0.0500,-0.0700,1.0000
C00596=18.250,-112.380,86.520,-0.1200,-0.0500,0.9900
C00597=16.720,-104.900,85.430,-0.1300,-0.0200,0.9900
C00598=15.480,-96.840,83.210,-0.1100,-0.0200,0.9900
C00599=14.350,-89.660,80.320,-0.0700,-0.0100,1.0000
C00600=13.160,-84.300,77.530,0.0100,0.0000,1.0000
C00601=11.120,-81.210,75.530,0.2600,0.3600,0.8900
C00602=6.930,-80.490,74.730,0.0300,0.6000,0.8000
C00603=3.190,-80.650,74.700,-0.0300,0.6100,0.7900
C00604=0.000,-80.700,74.720,-0.0000,0.6100,0.7900
C00605=0.000,-80.700,74.720,-0.0000,0.6100,0.7900
C00606=-3.190,-80.650,74.700,0.0300,0.6100,0.7900
C00607=-6.930,-80.490,74.730,-0.0300,0.6000,0.8000
C00608=-11.120,-81.210,75.530,-0.2600,0.3600,0.8900
C00609=-13.160,-84.300,77.530,-0.0100,0.0000,1.0000
C00610=-14.350,-89.660,80.320,0.0700,-0.0100,1.0000
C00611=-15.480,-96.840,83.210,0.1100,-0.0200,0.9900
C00612=-16.720,-104.900,85.430,0.1300,-0.0200,0.9900
C00613=-18.250,-112.380,86.520,0.1200,-0.0500,0.9900
C00614=-22.490,-117.840,87.100,0.0500,-0.0700,1.0000
C00615=-28.970,-120.420,87.570,0.0100,-0.0400,1.0000
C00616=-36.370,-119.540,88.050,-0.0000,-0.0000,1.0000
C00617=-44.010,-116.990,88.360,-0.0000,-0.0000,1.0000
C00618=-51.610,-113.840,88.360,-0.0000,-0.0000,1.0000
C00619=-58.810,-110.250,88.050,-0.0000,-0.0000,1.0000
C00620=-64.670,-105.630,87.570,-0.0300,-0.0300,1.0000
C00621=-67.420,-99.230,87.100,-0.0800,-0.0100,1.0000
C00622=-66.560,-92.380,86.520,-0.1200,0.0500,0.9900
C00623=-62.360,-86.000,85.430,-0.1100,0.0700,0.9900
C00624=-57.530,-79.420,83.210,-0.0900,0.0600,0.9900
C00625=-53.250,-73.540,80.320,-0.0600,0.0400,1.0000
C00626=-50.300,-68.910,77.530,0.0100,-0.0100,1.0000
C00627=-49.560,-65.290,75.530,0.4400,0.0700,0.8900
C00628=-52.020,-61.810,74.730,0.4500,0.4000,0.8000
C00629=-54.770,-59.280,74.700,0.4100,0.4500,0.7900
C00630=-57.070,-57.070,74.720,0.4300,0.4300,0.7900
C00631=-59.280,-54.770,74.700,0.4500,0.4100,0.7900
C00632=-61.810,-52.020,74.730,0.4000,0.4500,0.8000
C00633=-65.290,-49.560,75.530,0.0700,0.4400,0.8900
C00634=-68.910,-50.300,77.530,-0.0100,0.0100,1.0000
C00635=-73.540,-53.250,80.320,0.0400,-0.0600,1.0000
C00636=-79.420,-57.530,83.210,0.0600,-0.0900,0.9900
C00637=-86.000,-62.360,85.430,0.0700,-0.1100,0.9900
C00638=-92.380,-66.560,86.520,0.0500,-0.1200,0.9900
C00639=-99.230,-67.420,87.100,-0.0100,-0.0800,1.0000
C00640=-105.630,-64.670,87.570,-0.0300,-0.0300,1.0000
C00641=-110.250,-58.810,88.050,-0.0000,-0.0000,1.0000
C00642=-113.840,-51.610,88.360,-0.0000,-0.0000,1.0000
C00643=-116.990,-44.010,88.360,-0.0000,-0.0000,1.0000
C00644=-119.540,-36.370,88.050,-0.0000,-0.0000,1.0000
C00645=-120.420,-28.970,87.570,-0.0400,0.0100,1.0000
C00646=-117.840,-22.490,87.100,-0.0700,0.0500,1.0000
C00647=-112.380,-18.250,86.520,-0.0500,0.1200,0.9900
C00648=-104.900,-16.720,85.430,-0.0200,0.1300,0.9900
C00649=-96.840,-15.480,83.210,-0.0200,0.1100,0.9900
C00650=-89.660,-14.350,80.320,-0.0100,0.0700,1.0000
C00651=-84.300,-13.160,77.530,0.0000,-0.0100,1.0000
C00652=-81.210,-11.120,75.530,0.3600,-0.2600,0.8900
C00653=-80.490,-6.930,74.730,0.6000,-0.0300,0.8000
C00654=-80.650,-3.190,74.700,0.6100,0.0300,0.7900
C00655=-80.700,0.000,74.720,0.6100,0.0000,0.7900
C00656=-80.650,3.190,74.700,0.6100,-0.0300,0.7900
C00657=-80.490,6.930,74.730,0.6000,0.0300,0.8000
C00658=-81.210,11.120,75.530,0.3600,0.2600,0.8900
C00659=-84.300,13.160,77.530,0.0000,0.0100,1.0000
C00660=-89.660,14.350,80.320,-0.0100,-0.0700,1.0000
C00661=-96.840,15.480,83.210,-0.0200,-0.1100,0.9900
C00662=-104.900,16.720,85.430,-0.0200,-0.1300,0.9900
C00663=-112.380,18.250,86.520,-0.0500,-0.1200,0.9900
C00664=-117.840,22.490,87.100,-0.0700,-0.0500,1.0000
C00665=-120.420,28.970,87.570,-0.0400,-0.0100,1.0000
C00666=-119.540,36.370,88.050,-0.0000,0.0000,1.0000
C00667=-116.990,44.010,88.360,-0.0000,0.0000,1.0000
C00668=-113.840,51.610,88.360,-0.0000,0.0000,1.0000
C00669=-110.250,58.810,88.050,-0.0000,0.0000,1.0000
C00670=-105.630,64.670,87.570,-0.0300,0.0300,1.0000
C00671=-99.230,67.420,87.100,-0.0100,0.0800,1.0000
C00672=-92.380,66.560,86.520,0.0500,0.1200,0.9900
C00673=-86.000,62.360,85.430,0.0700,0.1100,0.9900
C00674=-79.420,57.530,83.210,0.0600,0.0900,0.9900
C00675=-73.540,53.250,80.320,0.0400,0.0600,1.0000
C00676=-68.910,50.300,77.530,-0.0100,-0.0100,1.0000
C00677=-65.290,49.560,75.530,0.0700,-0.4400,0.8900
C00678=-61.810,52.020,74.730,0.4000,-0.4500,0.8000
C00679=-59.280,54.770,74.700,0.4500,-0.4100,0.7900
C00680=-57.070,57.070,74.720,0.4300,-0.4300,0.7900
C00681=-54.770,59.280,74.700,0.4100,-0.4500,0.7900
C00682=-52.020,61.810,74.730,0.4500,-0.4000,0.8000
C00683=-49.560,65.290,75.530,0.4400,-0.0700,0.8900
C00684=-50.300,68.910,77.530,0.0100,0.0100,1.0000
C00685=-53.250,73.540,80.320,-0.0600,-0.0400,1.0000
C00686=-57.530,79.420,83.210,-0.0900,-0.0600,0.9900
C00687=-62.360,86.000,85.430,-0.1100,-0.0700,0.9900
C00688=-66.560,92.380,86.520,-0.1200,-0.0500,0.9900
C00689=-67.420,99.230,87.100,-0.0800,0.0100,1.0000
C00690=-64.670,105.630,87.570,-0.0300,0.0300,1.0000
C00691=-58.810,110.250,88.050,-0.0000,0.0000,1.0000
C00692=-51.610,113.840,88.360,-0.0000,0.0000,1.0000
C00693=-44.010,116.990,88.360,-0.0000,0.0000,1.0000
C00694=-36.370,119.540,88.050,-0.0000,0.0000,1.0000
C00695=-28.970,120.420,87.570,0.0100,0.0400,1.0000
C00696=-22.490,117.840,87.100,0.0500,0.0700,1.0000
C00697=-18.250,112.380,86.520,0.1200,0.0500,0.9900
C00698=-16.720,104.900,85.430,0.1300,0.0200,0.9900
C00699=-15.480,96.840,83.210,0.1100,0.0200,0.9900
C00700=-14.350,89.660,80.320,0.0700,0.0100,1.0000
C00701=-13.160,84.300,77.530,-0.0100,-0.0000,1.0000
C00702=-11.120,81.210,75.530,-0.2600,-0.3600,0.8900
C00703=-6.930,80.490,74.730,-0.0300,-0.6000,0.8000
C00704=-3.190,80.650,74.700,0.0300,-0.6100,0.7900
C00705=0.000,80.700,74.720,-0.0000,-0.6100,0.7900
C00706=0.000,79.670,76.070,-0.0000,-0.6000,0.8000
C00707=-3.100,79.620,76.050,0.0300,-0.6000,0.8000
C00708=-6.770,79.470,76.090,-0.0300,-0.5900,0.8000
C00709=-10.930,80.230,76.900,-0.2600,-0.3500,0.9000
C00710=-12.930,83.420,78.960,-0.0100,-0.0000,1.0000
C00711=-14.090,88.930,81.830,0.0700,0.0100,1.0000
C00712=-15.210,96.300,84.800,0.1100,0.0200,0.9900
C00713=-16.440,104.570,87.070,0.1300,0.0200,0.9900
C00714=-17.950,112.220,88.190,0.1200,0.0500,0.9900
C00715=-22.210,117.810,88.780,0.0500,0.0700,1.0000
C00716=-28.740,120.460,89.260,0.0100,0.0400,1.0000
C00717=-36.230,119.590,89.740,-0.0000,0.0000,1.0000
C00718=-43.960,117.010,90.060,-0.0000,0.0000,1.0000
C00719=-51.650,113.820,90.060,-0.0000,0.0000,1.0000
C00720=-58.940,110.180,89.740,-0.0000,0.0000,1.0000
C00721=-64.850,105.500,89.260,-0.0300,0.0200,1.0000
C00722=-67.600,99.010,88.780,-0.0800,0.0100,1.0000
C00723=-66.660,92.040,88.190,-0.1200,-0.0500,0.9900
C00724=-62.320,85.560,87.070,-0.1100,-0.0700,0.9900
C00725=-57.340,78.850,84.800,-0.0900,-0.0600,0.9900
C00726=-52.920,72.840,81.830,-0.0600,-0.0400,1.0000
C00727=-49.840,68.120,78.960,0.0100,0.0000,1.0000
C00728=-49.010,64.460,76.900,0.4300,-0.0600,0.9000
C00729=-51.410,60.980,76.090,0.4400,-0.4000,0.8000
C00730=-54.110,58.490,76.050,0.4100,-0.4500,0.8000
C00731=-56.340,56.340,76.070,0.4300,-0.4300,0.8000
C00732=-58.490,54.110,76.050,0.4500,-0.4100,0.8000
C00733=-60.980,51.410,76.090,0.4000,-0.4400,0.8000
C00734=-64.460,49.010,76.900,0.0600,-0.4300,0.9000
C00735=-68.120,49.840,78.960,-0.0000,-0.0100,1.0000
C00736=-72.840,52.920,81.830,0.0400,0.0600,1.0000
C00737=-78.850,57.340,84.800,0.0600,0.0900,0.9900
C00738=-85.560,62.320,87.070,0.0700,0.1100,0.9900
C00739=-92.040,66.660,88.190,0.0500,0.1200,0.9900
C00740=-99.010,67.600,88.780,-0.0100,0.0800,1.0000
C00741=-105.500,64.850,89.260,-0.0200,0.0300,1.0000
C00742=-110.180,58.940,89.740,-0.0000,0.0000,1.0000
C00743=-113.820,51.650,90.060,-0.0000,0.0000,1.0000
C00744=-117.010,43.960,90.060,-0.0000,0.0000,1.0000
C00745=-119.590,36.230,89.740,-0.0000,0.0000,1.0000
C00746=-120.460,28.740,89.260,-0.0400,-0.0100,1.0000
C00747=-117.810,22.210,88.780,-0.0700,-0.0500,1.0000
C00748=-112.220,17.950,88.190,-0.0500,-0.1200,0.9900
C00749=-104.570,16.440,87.070,-0.0200,-0.1300,0.9900
C00750=-96.300,15.210,84.800,-0.0200,-0.1100,0.9900
C00751=-88.930,14.090,81.830,-0.0100,-0.0700,1.0000
C00752=-83.420,12.930,78.960,0.0000,0.0100,1.0000
C00753=-80.230,10.930,76.900,0.3500,0.2600,0.9000
C00754=-79.470,6.770,76.090,0.5900,0.0300,0.8000
C00755=-79.620,3.100,76.050,0.6000,-0.0300,0.8000
C00756=-79.670,0.000,76.070,0.6000,0.0000,0.8000
C00757=-79.620,-3.100,76.050,0.6000,0.0300,0.8000
C00758=-79.470,-6.770,76.090,0.5900,-0.0300,0.8000
C00759=-80.230,-10.930,76.900,0.3500,-0.2600,0.9000
C00760=-83.420,-12.930,78.960,0.0000,-0.0100,1.0000
C00761=-88.930,-14.090,81.830,-0.0100,0.0700,1.0000
C00762=-96.300,-15.210,84.800,-0.0200,0.1100,0.9900
C00763=-104.570,-16.440,87.070,-0.0200,0.1300,0.9900
C00764=-112.220,-17.950,88.190,-0.0500,0.1200,0.9900
C00765=-117.810,-22.210,88.780,-0.0700,0.0500,1.0000
C00766=-120.460,-28.740,89.260,-0.0400,0.0100,1.0000
C00767=-119.590,-36.230,89.740,-0.0000,-0.0000,1.0000
C00768=-117.010,-43.960,90.060,-0.0000,-0.0000,1.0000
C00769=-113.820,-51.650,90.060,-0.0000,-0.0000,1.0000
C00770=-110.180,-58.940,89.740,-0.0000,-0.0000,1.0000
C00771=-105.500,-64.850,89.260,-0.0200,-0.0300,1.0000
C00772=-99.010,-67.600,88.780,-0.0100,-0.0800,1.0000
C00773=-92.040,-66.660,88.190,0.0500,-0.1200,0.9900
C00774=-85.560,-62.320,87.070,0.0700,-0.1100,0.9900
C00775=-78.850,-57.340,84.800,0.0600,-0.0900,0.9900
C00776=-72.840,-52.920,81.830,0.0400,-0.0600,1.0000
C00777=-68.120,-49.840,78.960,-0.0000,0.0100,1.0000
C00778=-64.460,-49.010,76.900,0.0600,0.4300,0.9000
C00779=-60.980,-51.410,76.090,0.4000,0.4400,0.8000
C00780=-58.490,-54.110,76.050,0.4500,0.4100,0.8000
C00781=-56.340,-56.340,76.070,0.4300,0.4300,0.8000
C00782=-54.110,-58.490,76.050,0.4100,0.4500,0.8000
C00783=-51.410,-60.980,76.090,0.4400,0.4000,0.8000
C00784=-49.010,-64.460,76.900,0.4300,0.0600,0.9000
C00785=-49.840,-68.120,78.960,0.0100,-0.0000,1.0000
C00786=-52.920,-72.840,81.830,-0.0600,0.0400,1.0000
C00787=-57.340,-78.850,84.800,-0.0900,0.0600,0.9900
C00788=-62.320,-85.560,87.070,-0.1100,0.0700,0.9900
C00789=-66.660,-92.040,88.190,-0.1200,0.0500,0.9900
C00790=-67.600,-99.010,88.780,-0.0800,-0.0100,1.0000
C00791=-64.850,-105.500,89.260,-0.0300,-0.0200,1.0000
C00792=-58.940,-110.180,89.740,-0.0000,-0.0000,1.0000
C00793=-51.650,-113.820,90.060,-0.0000,-0.0000,1.0000
C00794=-43.960,-117.010,90.060,-0.0000,-0.0000,1.0000
C00795=-36.230,-119.590,89.740,-0.0000,-0.0000,1.0000
C00796=-28.740,-120.460,89.260,0.0100,-0.0400,1.0000
C00797=-22.210,-117.810,88.780,0.0500,-0.0700,1.0000
C00798=-17.950,-112.220,88.190,0.1200,-0.0500,0.9900
C00799=-16.440,-104.570,87.070,0.1300,-0.0200,0.9900
C00800=-15.210,-96.300,84.800,0.1100,-0.0200,0.9900
C00801=-14.090,-88.930,81.830,0.0700,-0.0100,1.0000
C00802=-12.930,-83.420,78.960,-0.0100,0.0000,1.0000
C00803=-10.930,-80.230,76.900,-0.2600,0.3500,0.9000
C00804=-6.770,-79.470,76.090,-0.0300,0.5900,0.8000
C00805=-3.100,-79.620,76.050,0.0300,0.6000,0.8000
C00806=0.000,-79.670,76.070,-0.0000,0.6000,0.8000
C00807=0.000,-79.670,76.070,-0.0000,0.6000,0.8000
C00808=3.100,-79.620,76.050,-0.0300,0.6000,0.8000
C00809=6.770,-79.470,76.090,0.0300,0.5900,0.8000
C00810=10.930,-80.230,76.900,0.2600,0.3500,0.9000
C00811=12.930,-83.420,78.960,0.0100,0.0000,1.0000
C00812=14.090,-88.930,81.830,-0.0700,-0.0100,1.0000
C00813=15.210,-96.300,84.800,-0.1100,-0.0200,0.9900
C00814=16.440,-104.570,87.070,-0.1300,-0.0200,0.9900
C00815=17.950,-112.220,88.190,-0.1200,-0.0500,0.9900
C00816=22.210,-117.810,88.780,-0.0500,-0.0700,1.0000
C00817=28.740,-120.460,89.260,-0.0100,-0.0400,1.0000
C00818=36.230,-119.590,89.740,0.0000,-0.0000,1.0000
C00819=43.960,-117.010,90.060,0.0000,-0.0000,1.0000
C00820=51.650,-113.820,90.060,0.0000,-0.0000,1.0000
C00821=58.940,-110.180,89.740,0.0000,-0.0000,1.0000
C00822=64.850,-105.500,89.260,0.0300,-0.0200,1.0000
C00823=67.600,-99.010,88.780,0.0800,-0.0100,1.0000
C00824=66.660,-92.040,88.190,0.1200,0.0500,0.9900
C00825=62.320,-85.560,87.070,0.1100,0.0700,0.9900
C00826=57.340,-78.850,84.800,0.0900,0.0600,0.9900
C00827=52.920,-72.840,81.830,0.0600,0.0400,1.0000
C00828=49.840,-68.120,78.960,-0.0100,-0.0000,1.0000
C00829=49.010,-64.460,76.900,-0.4300,0.0600,0.9000
C00830=51.410,-60.980,76.090,-0.4400,0.4000,0.8000
C00831=54.110,-58.490,76.050,-0.4100,0.4500,0.8000
C00832=56.340,-56.340,76.070,-0.4300,0.4300,0.8000
C00833=58.490,-54.110,76.050,-0.4500,0.4100,0.8000
C00834=60.980,-51.410,76.090,-0.4000,0.4400,0.8000
C00835=64.460,-49.010,76.900,-0.0600,0.4300,0.9000
C00836=68.120,-49.840,78.960,0.0000,0.0100,1.0000
C00837=72.840,-52.920,81.830,-0.0400,-0.0600,1.0000
C00838=78.850,-57.340,84.800,-0.0600,-0.0900,0.9900
C00839=85.560,-62.320,87.070,-0.0700,-0.1100,0.9900
C00840=92.040,-66.660,88.190,-0.0500,-0.1200,0.9900
C00841=99.010,-67.600,88.780,0.0100,-0.0800,1.0000
C00842=105.500,-64.850,89.260,0.0200,-0.0300,1.0000
C00843=110.180,-58.940,89.740,0.0000,-0.0000,1.0000
C00844=113.820,-51.650,90.060,0.0000,-0.0000,1.0000
C00845=117.010,-43.960,90.060,0.0000,-0.0000,1.0000
C00846=119.590,-36.230,89.740,0.0000,-0.0000,1.0000
C00847=120.460,-28.740,89.260,0.0400,0.0100,1.0000
C00848=117.810,-22.210,88.780,0.0700,0.0500,1.0000
C00849=112.220,-17.950,88.190,0.0500,0.1200,0.9900
C00850=104.570,-16.440,87.070,0.0200,0.1300,0.9900
C00851=96.300,-15.210,84.800,0.0200,0.1100,0.9900
C00852=88.930,-14.090,81.830,0.0100,0.0700,1.0000
C00853=83.420,-12.930,78.960,-0.0000,-0.0100,1.0000
C00854=80.230,-10.930,76.900,-0.3500,-0.2600,0.9000
C00855=79.470,-6.770,76.090,-0.5900,-0.0300,0.8000
C00856=79.620,-3.100,76.050,-0.6000,0.0300,0.8000
C00857=79.670,0.000,76.070,-0.6000,-0.0000,0.8000
C00858=79.620,3.100,76.050,-0.6000,-0.0300,0.8000
C00859=79.470,6.770,76.090,-0.5900,0.0300,0.8000
C00860=80.230,10.930,76.900,-0.3500,0.2600,0.9000
C00861=83.420,12.930,78.960,-0.0000,0.0100,1.0000
C00862=88.930,14.090,81.830,0.0100,-0.0700,1.0000
C00863=96.300,15.210,84.800,0.0200,-0.1100,0.9900
C00864=104.570,16.440,87.070,0.0200,-0.1300,0.9900
C00865=112.220,17.950,88.190,0.0500,-0.1200,0.9900
C00866=117.810,22.210,88.780,0.0700,-0.0500,1.0000
C00867=120.460,28.740,89.260,0.0400,-0.0100,1.0000
C00868=119.590,36.230,89.740,0.0000,0.0000,1.0000
C00869=117.010,43.960,90.060,0.0000,0.0000,1.0000
C00870=113.820,51.650,90.060,0.0000,0.0000,1.0000
C00871=110.180,58.940,89.740,0.0000,0.0000,1.0000
C00872=105.500,64.850,89.260,0.0200,0.0300,1.0000
C00873=99.010,67.600,88.780,0.0100,0.0800,1.0000
C00874=92.040,66.660,88.190,-0.0500,0.1200,0.9900
C00875=85.560,62.320,87.070,-0.0700,0.1100,0.9900
C00876=78.850,57.340,84.800,-0.0600,0.0900,0.9900
C00877=72.840,52.920,81.830,-0.0400,0.0600,1.0000
C00878=68.120,49.840,78.960,0.0000,-0.0100,1.0000
C00879=64.460,49.010,76.900,-0.0600,-0.4300,0.9000
C00880=60.980,51.410,76.090,-0.4000,-0.4400,0.8000
C00881=58.490,54.110,76.050,-0.4500,-0.4100,0.8000
C00882=56.340,56.340,76.070,-0.4300,-0.4300,0.8000
C00883=54.110,58.490,76.050,-0.4100,-0.4500,0.8000
C00884=51.410,60.980,76.090,-0.4400,-0.4000,0.8000
C00885=49.010,64.460,76.900,-0.4300,-0.0600,0.9000
C00886=49.840,68.120,78.960,-0.0100,0.0000,1.0000
C00887=52.920,72.840,81.830,0.0600,-0.0400,1.0000
C00888=57.340,78.850,84.800,0.0900,-0.0600,0.9900
C00889=62.320,85.560,87.070,0.1100,-0.0700,0.9900
C00890=66.660,92.040,88.190,0.1200,-0.0500,0.9900
C00891=67.600,99.010,88.780,0.0800,0.0100,1.0000
C00892=64.850,105.500,89.260,0.0300,0.0200,1.0000
C00893=58.940,110.180,89.740,0.0000,0.0000,1.0000
C00894=51.650,113.820,90.060,0.0000,0.0000,1.0000
C00895=43.960,117.010,90.060,0.0000,0.0000,1.0000
C00896=36.230,119.590,89.740,0.0000,0.0000,1.0000
C00897=28.740,120.460,89.260,-0.0100,0.0400,1.0000
C00898=22.210,117.810,88.780,-0.0500,0.0700,1.0000
C00899=17.950,112.220,88.190,-0.1200,0.0500,0.9900
C00900=16.440,104.570,87.070,-0.1300,0.0200,0.9900
C00901=15.210,96.300,84.800,-0.1100,0.0200,0.9900
C00902=14.090,88.930,81.830,-0.0700,0.0100,1.0000
C00903=12.930,83.420,78.960,0.0100,-0.0000,1.0000
C00904=10.930,80.230,76.900,0.2600,-0.3500,0.9000
C00905=6.770,79.470,76.090,0.0300,-0.5900,0.8000
C00906=3.100,79.620,76.050,-0.0300,-0.6000,0.8000
C00907=0.000,79.670,76.070,-0.0000,-0.6000,0.8000
C00908=0.000,78.650,77.430,-0.0000,-0.6000,0.8000
C00909=3.010,78.600,77.410,-0.0300,-0.6000,0.8000
C00910=6.610,78.460,77.450,0.0400,-0.5900,0.8100
C00911=10.730,79.260,78.280,0.2600,-0.3300,0.9100
C00912=12.700,82.550,80.410,0.0000,-0.0000,1.0000
C00913=13.830,88.220,83.350,-0.0700,0.0100,1.0000
C00914=14.940,95.780,86.390,-0.1000,0.0200,0.9900
C00915=16.160,104.240,88.710,-0.1300,0.0200,0.9900
C00916=17.660,112.060,89.850,-0.1200,0.0500,0.9900
C00917=21.940,117.770,90.450,-0.0500,0.0600,1.0000
C00918=28.530,120.500,90.940,-0.0100,0.0400,1.0000
C00919=36.100,119.630,91.430,0.0000,0.0000,1.0000
C00920=43.920,117.030,91.760,0.0000,0.0000,1.0000
C00921=51.700,113.800,91.760,0.0000,0.0000,1.0000
C00922=59.070,110.120,91.430,0.0000,0.0000,1.0000
C00923=65.030,105.380,90.940,0.0300,0.0200,1.0000
C00924=67.770,98.790,90.450,0.0800,0.0100,1.0000
C00925=66.750,91.720,89.850,0.1200,-0.0500,0.9900
C00926=62.280,85.130,88.710,0.1000,-0.0700,0.9900
C00927=57.160,78.290,86.390,0.0900,-0.0600,0.9900
C00928=52.600,72.160,83.350,0.0600,-0.0400,1.0000
C00929=49.390,67.350,80.410,-0.0000,0.0000,1.0000
C00930=48.460,63.640,78.280,-0.4200,-0.0500,0.9100
C00931=50.810,60.160,77.450,-0.4400,-0.3900,0.8100
C00932=53.450,57.700,77.410,-0.4000,-0.4400,0.8000
C00933=55.620,55.620,77.430,-0.4200,-0.4200,0.8000
C00934=57.700,53.450,77.410,-0.4400,-0.4000,0.8000
C00935=60.160,50.810,77.450,-0.3900,-0.4400,0.8100
C00936=63.640,48.460,78.280,-0.0500,-0.4200,0.9100
C00937=67.350,49.390,80.410,0.0000,-0.0000,1.0000
C00938=72.160,52.600,83.350,-0.0400,0.0600,1.0000
C00939=78.290,57.160,86.390,-0.0600,0.0900,0.9900
C00940=85.130,62.280,88.710,-0.0700,0.1000,0.9900
C00941=91.720,66.750,89.850,-0.0500,0.1200,0.9900
C00942=98.790,67.770,90.450,0.0100,0.0800,1.0000
C00943=105.380,65.030,90.940,0.0200,0.0300,1.0000
C00944=110.120,59.070,91.430,0.0000,0.0000,1.0000
C00945=113.800,51.700,91.760,0.0000,0.0000,1.0000
C00946=117.030,43.920,91.760,0.0000,0.0000,1.0000
C00947=119.630,36.100,91.430,0.0000,0.0000,1.0000
C00948=120.500,28.530,90.940,0.0400,-0.0100,1.0000
C00949=117.770,21.940,90.450,0.0600,-0.0500,1.0000
C00950=112.060,17.660,89.850,0.0500,-0.1200,0.9900
C00951=104.240,16.160,88.710,0.0200,-0.1300,0.9900
C00952=95.780,14.940,86.390,0.0200,-0.1000,0.9900
C00953=88.220,13.830,83.350,0.0100,-0.0700,1.0000
C00954=82.550,12.700,80.410,-0.0000,0.0000,1.0000
C00955=79.260,10.730,78.280,-0.3300,0.2600,0.9100
C00956=78.460,6.610,77.450,-0.5900,0.0400,0.8100
C00957=78.600,3.010,77.410,-0.6000,-0.0300,0.8000
C00958=78.650,0.000,77.430,-0.6000,-0.0000,0.8000
C00959=78.600,-3.010,77.410,-0.6000,0.0300,0.8000
C00960=78.460,-6.610,77.450,-0.5900,-0.0400,0.8100
C00961=79.260,-10.730,78.280,-0.3300,-0.2600,0.9100
C00962=82.550,-12.700,80.410,-0.0000,-0.0000,1.0000
C00963=88.220,-13.830,83.350,0.0100,0.0700,1.0000
C00964=95.780,-14.940,86.390,0.0200,0.1000,0.9900
C00965=104.240,-16.160,88.710,0.0200,0.1300,0.9900
C00966=112.060,-17.660,89.850,0.0500,0.1200,0.9900
C00967=117.770,-21.940,90.450,0.0600,0.0500,1.0000
C00968=120.500,-28.530,90.940,0.0400,0.0100,1.0000
C00969=119.630,-36.100,91.430,0.0000,-0.0000,1.0000
C00970=117.030,-43.920,91.760,0.0000,-0.0000,1.0000
C00971=113.800,-51.700,91.760,0.0000,-0.0000,1.0000
C00972=110.120,-59.070,91.430,0.0000,-0.0000,1.0000
C00973=105.380,-65.030,90.940,0.0200,-0.0300,1.0000
C00974=98.790,-67.770,90.450,0.0100,-0.0800,1.0000
C00975=91.720,-66.750,89.850,-0.0500,-0.1200,0.9900
C00976=85.130,-62.280,88.710,-0.0700,-0.1000,0.9900
C00977=78.290,-57.160,86.390,-0.0600,-0.0900,0.9900
C00978=72.160,-52.600,83.350,-0.0400,-0.0600,1.0000
C00979=67.350,-49.390,80.410,0.0000,0.0000,1.0000
C00980=63.640,-48.460,78.280,-0.0500,0.4200,0.9100
C00981=60.160,-50.810,77.450,-0.3900,0.4400,0.8100
C00982=57.700,-53.450,77.410,-0.4400,0.4000,0.8000
C00983=55.620,-55.620,77.430,-0.4200,0.4200,0.8000
C00984=53.450,-57.700,77.410,-0.4000,0.4400,0.8000
C00985=50.810,-60.160,77.450,-0.4400,0.3900,0.8100
C00986=48.460,-63.640,78.280,-0.4200,0.0500,0.9100
C00987=49.390,-67.350,80.410,-0.0000,-0.0000,1.0000
C00988=52.600,-72.160,83.350,0.0600,0.0400,1.0000
C00989=57.160,-78.290,86.390,0.0900,0.0600,0.9900
C00990=62.280,-85.130,88.710,0.1000,0.0700,0.9900
C00991=66.750,-91.720,89.850,0.1200,0.0500,0.9900
C00992=67.770,-98.790,90.450,0.0800,-0.0100,1.0000
C00993=65.030,-105.380,90.940,0.0300,-0.0200,1.0000
C00994=59.070,-110.120,91.430,0.0000,-0.0000,1.0000
C00995=51.700,-113.800,91.760,0.0000,-0.0000,1.0000
C00996=43.920,-117.030,91.760,0.0000,-0.0000,1.0000
C00997=36.100,-119.630,91.430,0.0000,-0.0000,1.0000
C00998=28.530,-120.500,90.940,-0.0100,-0.0400,1.0000
C00999=21.940,-117.770,90.450,-0.0500,-0.0600,1.0000
C01000=17.660,-112.060,89.850,-0.1200,-0.0500,0.9900
C01001=16.160,-104.240,88.710,-0.1300,-0.0200,0.9900
C01002=14.940,-95.780,86.390,-0.1000,-0.0200,0.9900
C01003=13.830,-88.220,83.350,-0.0700,-0.0100,1.0000
C01004=12.700,-82.550,80.410,0.0000,0.0000,1.0000
C01005=10.730,-79.260,78.280,0.2600,0.3300,0.9100
C01006=6.610,-78.460,77.450,0.0400,0.5900,0.8100
C01007=3.010,-78.600,77.410,-0.0300,0.6000,0.8000
C01008=0.000,-78.650,77.430,-0.0000,0.6000,0.8000
C01009=0.000,-78.650,77.430,-0.0000,0.6000,0.8000
C01010=-3.010,-78.600,77.410,0.0300,0.6000,0.8000
C01011=-6.610,-78.460,77.450,-0.0400,0.5900,0.8100
C01012=-10.730,-79.260,78.280,-0.2600,0.3300,0.9100
C01013=-12.700,-82.550,80.410,-0.0000,0.0000,1.0000
C01014=-13.830,-88.220,83.350,0.0700,-0.0100,1.0000
C01015=-14.940,-95.780,86.390,0.1000,-0.0200,0.9900
C01016=-16.160,-104.240,88.710,0.1300,-0.0200,0.9900
C01017=-17.660,-112.060,89.850,0.1200,-0.0500,0.9900
C01018=-21.940,-117.770,90.450,0.0500,-0.0600,1.0000
C01019=-28.530,-120.500,90.940,0.0100,-0.0400,1.0000
C01020=-36.100,-119.630,91.430,-0.0000,-0.0000,1.0000
C01021=-43.920,-117.030,91.760,-0.0000,-0.0000,1.0000
C01022=-51.700,-113.800,91.760,-0.0000,-0.0000,1.0000
C01023=-59.070,-110.120,91.430,-0.0000,-0.0000,1.0000
C01024=-65.030,-105.380,90.940,-0.0300,-0.0200,1.0000
C01025=-67.770,-98.790,90.450,-0.0800,-0.0100,1.0000
C01026=-66.750,-91.720,89.850,-0.1200,0.0500,0.9900
C01027=-62.280,-85.130,88.710,-0.1000,0.0700,0.9900
C01028=-57.160,-78.290,86.390,-0.0900,0.0600,0.9900
C01029=-52.600,-72.160,83.350,-0.0600,0.0400,1.0000
C01030=-49.390,-67.350,80.410,0.0000,-0.0000,1.0000
C01031=-48.460,-63.640,78.280,0.4200,0.0500,0.9100
C01032=-50.810,-60.160,77.450,0.4400,0.3900,0.8100
C01033=-53.450,-57.700,77.410,0.4000,0.4400,0.8000
C01034=-55.620,-55.620,77.430,0.4200,0.4200,0.8000
C01035=-57.700,-53.450,77.410,0.4400,0.4000,0.8000
C01036=-60.160,-50.810,77.450,0.3900,0.4400,0.8100
C01037=-63.640,-48.460,78.280,0.0500,0.4200,0.9100
C01038=-67.350,-49.390,80.410,-0.0000,0.0000,1.0000
C01039=-72.160,-52.600,83.350,0.0400,-0.0600,1.0000
C01040=-78.290,-57.160,86.390,0.0600,-0.0900,0.9900
C01041=-85.130,-62.280,88.710,0.0700,-0.1000,0.9900
C01042=-91.720,-66.750,89.850,0.0500,-0.1200,0.9900
C01043=-98.790,-67.770,90.450,-0.0100,-0.0800,1.0000
C01044=-105.380,-65.030,90.940,-0.0200,-0.0300,1.0000
C01045=-110.120,-59.070,91.430,-0.0000,-0.0000,1.0000
C01046=-113.800,-51.700,91.760,-0.0000,-0.0000,1.0000
C01047=-117.030,-43.920,91.760,-0.0000,-0.0000,1.0000
C01048=-119.630,-36.100,91.430,-0.0000,-0.0000,1.0000
C01049=-120.500,-28.530,90.940,-0.0400,0.0100,1.0000
C01050=-117.770,-21.940,90.450,-0.0600,0.0500,1.0000
C01051=-112.060,-17.660,89.850,-0.0500,0.1200,0.9900
C01052=-104.240,-16.160,88.710,-0.0200,0.1300,0.9900
C01053=-95.780,-14.940,86.390,-0.0200,0.1000,0.9900
C01054=-88.220,-13.830,83.350,-0.0100,0.0700,1.0000
C01055=-82.550,-12.700,80.410,0.0000,-0.0000,1.0000
C01056=-79.260,-10.730,78.280,0.3300,-0.2600,0.9100
C01057=-78.460,-6.610,77.450,0.5900,-0.0400,0.8100
C01058=-78.600,-3.010,77.410,0.6000,0.0300,0.8000
C01059=-78.650,0.000,77.430,0.6000,0.0000,0.8000
C01060=-78.600,3.010,77.410,0.6000,-0.0300,0.8000
C01061=-78.460,6.610,77.450,0.5900,0.0400,0.8100
C01062=-79.260,10.730,78.280,0.3300,0.2600,0.9100
C01063=-82.550,12.700,80.410,0.0000,0.0000,1.0000
C01064=-88.220,13.830,83.350,-0.0100,-0.0700,1.0000
C01065=-95.780,14.940,86.390,-0.0200,-0.1000,0.9900
C01066=-104.240,16.160,88.710,-0.0200,-0.1300,0.9900
C01067=-112.060,17.660,89.850,-0.0500,-0.1200,0.9900
C01068=-117.770,21.940,90.450,-0.0600,-0.0500,1.0000
C01069=-120.500,28.530,90.940,-0.0400,-0.0100,1.0000
C01070=-119.630,36.100,91.430,-0.0000,0.0000,1.0000
C01071=-117.030,43.920,91.760,-0.0000,0.0000,1.0000
C01072=-113.800,51.700,91.760,-0.0000,0.0000,1.0000
C01073=-110.120,59.070,91.430,-0.0000,0.0000,1.0000
C01074=-105.380,65.030,90.940,-0.0200,0.0300,1.0000
C01075=-98.790,67.770,90.450,-0.0100,0.0800,1.0000
C01076=-91.720,66.750,89.850,0.0500,0.1200,0.9900
C01077=-85.130,62.280,88.710,0.0700,0.1000,0.9900
C01078=-78.290,57.160,86.390,0.0600,0.0900,0.9900
C01079=-72.160,52.600,83.350,0.0400,0.0600,1.0000
C01080=-67.350,49.390,80.410,-0.0000,-0.0000,1.0000
C01081=-63.640,48.460,78.280,0.0500,-0.4200,0.9100
C01082=-60.160,50.810,77.450,0.3900,-0.4400,0.8100
C01083=-57.700,53.450,77.410,0.4400,-0.4000,0.8000
C01084=-55.620,55.620,77.430,0.4200,-0.4200,0.8000
C01085=-53.450,57.700,77.410,0.4000,-0.4400,0.8000
C01086=-50.810,60.160,77.450,0.4400,-0.3900,0.8100
C01087=-48.460,63.640,78.280,0.4200,-0.0500,0.9100
C01088=-49.390,67.350,80.410,0.0000,0.0000,1.0000
C01089=-52.600,72.160,83.350,-0.0600,-0.0400,1.0000
C01090=-57.160,78.290,86.390,-0.0900,-0.0600,0.9900
C01091=-62.280,85.130,88.710,-0.1000,-0.0700,0.9900
C01092=-66.750,91.720,89.850,-0.1200,-0.0500,0.9900
C01093=-67.770,98.790,90.450,-0.0800,0.0100,1.0000
C01094=-65.030,105.380,90.940,-0.0300,0.0200,1.0000
C01095=-59.070,110.120,91.430,-0.0000,0.0000,1.0000
C01096=-51.700,113.800,91.760,-0.0000,0.0000,1.0000
C01097=-43.920,117.030,91.760,-0.0000,0.0000,1.0000
C01098=-36.100,119.630,91.430,-0.0000,0.0000,1.0000
C01099=-28.530,120.500,90.940,0.0100,0.0400,1.0000
C01100=-21.940,117.770,90.450,0.0500,0.0600,1.0000
C01101=-17.660,112.060,89.850,0.1200,0.0500,0.9900
C01102=-16.160,104.240,88.710,0.1300,0.0200,0.9900
C01103=-14.940,95.780,86.390,0.1000,0.0200,0.9900
C01104=-13.830,88.220,83.350,0.0700,0.0100,1.0000
C01105=-12.700,82.550,80.410,-0.0000,-0.0000,1.0000
C01106=-10.730,79.260,78.280,-0.2600,-0.3300,0.9100
C01107=-6.610,78.460,77.450,-0.0400,-0.5900,0.8100
C01108=-3.010,78.600,77.410,0.0300,-0.6000,0.8000
C01109=0.000,78.650,77.430,-0.0000,-0.6000,0.8000
C01110=0.000,77.640,78.800,-0.0000,-0.5900,0.8100
C01111=-2.910,77.590,78.770,0.0300,-0.5900,0.8100
C01112=-6.460,77.460,78.810,-0.0400,-0.5800,0.8100
C01113=-10.550,78.300,79.670,-0.2600,-0.3200,0.9100
C01114=-12.470,81.690,81.850,0.0100,0.0000,1.0000
C01115=-13.580,87.510,84.880,0.0700,0.0100,1.0000
C01116=-14.680,95.270,87.990,0.1000,0.0200,0.9900
C01117=-15.890,103.920,90.360,0.1200,0.0200,0.9900
C01118=-17.370,111.900,91.520,0.1200,0.0400,0.9900
C01119=-21.670,117.740,92.130,0.0500,0.0600,1.0000
C01120=-28.320,120.530,92.630,0.0100,0.0400,1.0000
C01121=-35.970,119.670,93.130,-0.0000,0.0000,1.0000
C01122=-43.870,117.040,93.460,-0.0000,0.0000,1.0000
C01123=-51.740,113.790,93.460,-0.0000,0.0000,1.0000
C01124=-59.190,110.060,93.130,-0.0000,0.0000,1.0000
C01125=-65.200,105.260,92.630,-0.0300,0.0200,1.0000
C01126=-67.930,98.580,92.130,-0.0800,0.0100,1.0000
C01127=-66.840,91.410,91.520,-0.1100,-0.0500,0.9900
C01128=-62.240,84.720,90.360,-0.1000,-0.0700,0.9900
C01129=-56.980,77.740,87.990,-0.0900,-0.0600,0.9900
C01130=-52.280,71.480,84.880,-0.0600,-0.0400,1.0000
C01131=-48.950,66.580,81.850,-0.0100,-0.0000,1.0000
C01132=-47.910,62.820,79.670,0.4100,-0.0500,0.9100
C01133=-50.210,59.340,78.810,0.4400,-0.3800,0.8100
C01134=-52.810,56.920,78.770,0.4000,-0.4400,0.8100
C01135=-54.900,54.900,78.800,0.4200,-0.4200,0.8100
C01136=-56.920,52.810,78.770,0.4400,-0.4000,0.8100
C01137=-59.340,50.210,78.810,0.3800,-0.4400,0.8100
C01138=-62.820,47.910,79.670,0.0500,-0.4100,0.9100
C01139=-66.580,48.950,81.850,0.0000,0.0100,1.0000
C01140=-71.480,52.280,84.880,0.0400,0.0600,1.0000
C01141=-77.740,56.980,87.990,0.0600,0.0900,0.9900
C01142=-84.720,62.240,90.360,0.0700,0.1000,0.9900
C01143=-91.410,66.840,91.520,0.0500,0.1100,0.9900
C01144=-98.580,67.930,92.130,-0.0100,0.0800,1.0000
C01145=-105.260,65.200,92.630,-0.0200,0.0300,1.0000
C01146=-110.060,59.190,93.130,-0.0000,0.0000,1.0000
C01147=-113.790,51.740,93.460,-0.0000,0.0000,1.0000
C01148=-117.040,43.870,93.460,-0.0000,0.0000,1.0000
C01149=-119.670,35.970,93.130,-0.0000,0.0000,1.0000
C01150=-120.530,28.320,92.630,-0.0400,-0.0100,1.0000
C01151=-117.740,21.670,92.130,-0.0600,-0.0500,1.0000
C01152=-111.900,17.370,91.520,-0.0400,-0.1200,0.9900
C01153=-103.920,15.890,90.360,-0.0200,-0.1200,0.9900
C01154=-95.270,14.680,87.990,-0.0200,-0.1000,0.9900
C01155=-87.510,13.580,84.880,-0.0100,-0.0700,1.0000
C01156=-81.690,12.470,81.850,-0.0000,-0.0100,1.0000
C01157=-78.300,10.550,79.670,0.3200,0.2600,0.9100
C01158=-77.460,6.460,78.810,0.5800,0.0400,0.8100
C01159=-77.590,2.910,78.770,0.5900,-0.0300,0.8100
C01160=-77.640,0.000,78.800,0.5900,0.0000,0.8100
C01161=-77.590,-2.910,78.770,0.5900,0.0300,0.8100
C01162=-77.460,-6.460,78.810,0.5800,-0.0400,0.8100
C01163=-78.300,-10.550,79.670,0.3200,-0.2600,0.9100
C01164=-81.690,-12.470,81.850,-0.0000,0.0100,1.0000
C01165=-87.510,-13.580,84.880,-0.0100,0.0700,1.0000
C01166=-95.270,-14.680,87.990,-0.0200,0.1000,0.9900
C01167=-103.920,-15.890,90.360,-0.0200,0.1200,0.9900
C01168=-111.900,-17.370,91.520,-0.0400,0.1200,0.9900
C01169=-117.740,-21.670,92.130,-0.0600,0.0500,1.0000
C01170=-120.530,-28.320,92.630,-0.0400,0.0100,1.0000
C01171=-119.670,-35.970,93.130,-0.0000,-0.0000,1.0000
C01172=-117.040,-43.870,93.460,-0.0000,-0.0000,1.0000
C01173=-113.790,-51.740,93.460,-0.0000,-0.0000,1.0000
C01174=-110.060,-59.190,93.130,-0.0000,-0.0000,1.0000
C01175=-105.260,-65.200,92.630,-0.0200,-0.0300,1.0000
C01176=-98.580,-67.930,92.130,-0.0100,-0.0800,1.0000
C01177=-91.410,-66.840,91.520,0.0500,-0.1100,0.9900
C01178=-84.720,-62.240,90.360,0.0700,-0.1000,0.9900
C01179=-77.740,-56.980,87.990,0.0600,-0.0900,0.9900
C01180=-71.480,-52.280,84.880,0.0400,-0.0600,1.0000
C01181=-66.580,-48.950,81.850,0.0000,-0.0100,1.0000
C01182=-62.820,-47.910,79.670,0.0500,0.4100,0.9100
C01183=-59.340,-50.210,78.810,0.3800,0.4400,0.8100
C01184=-56.920,-52.810,78.770,0.4400,0.4000,0.8100
C01185=-54.900,-54.900,78.800,0.4200,0.4200,0.8100
C01186=-52.810,-56.920,78.770,0.4000,0.4400,0.8100
C01187=-50.210,-59.340,78.810,0.4400,0.3800,0.8100
C01188=-47.910,-62.820,79.670,0.4100,0.0500,0.9100
C01189=-48.950,-66.580,81.850,-0.0100,0.0000,1.0000
C01190=-52.280,-71.480,84.880,-0.0600,0.0400,1.0000
C01191=-56.980,-77.740,87.990,-0.0900,0.0600,0.9900
C01192=-62.240,-84.720,90.360,-0.1000,0.0700,0.9900
C01193=-66.840,-91.410,91.520,-0.1100,0.0500,0.9900
C01194=-67.930,-98.580,92.130,-0.0800,-0.0100,1.0000
C01195=-65.200,-105.260,92.630,-0.0300,-0.0200,1.0000
C01196=-59.190,-110.060,93.130,-0.0000,-0.0000,1.0000
C01197=-51.740,-113.790,93.460,-0.0000,-0.0000,1.0000
C01198=-43.870,-117.040,93.460,-0.0000,-0.0000,1.0000
C01199=-35.970,-119.670,93.130,-0.0000,-0.0000,1.0000
C01200=-28.320,-120.530,92.630,0.0100,-0.0400,1.0000
C01201=-21.670,-117.740,92.130,0.0500,-0.0600,1.0000
C01202=-17.370,-111.900,91.520,0.1200,-0.0400,0.9900
C01203=-15.890,-103.920,90.360,0.1200,-0.0200,0.9900
C01204=-14.680,-95.270,87.990,0.1000,-0.0200,0.9900
C01205=-13.580,-87.510,84.880,0.0700,-0.0100,1.0000
C01206=-12.470,-81.690,81.850,0.0100,-0.0000,1.0000
C01207=-10.550,-78.300,79.670,-0.2600,0.3200,0.9100
C01208=-6.460,-77.460,78.810,-0.0400,0.5800,0.8100
C01209=-2.910,-77.590,78.770,0.0300,0.5900,0.8100
C01210=0.000,-77.640,78.800,-0.0000,0.5900,0.8100
C01211=0.000,-77.640,78.800,-0.0000,0.5900,0.8100
C01212=2.910,-77.590,78.770,-0.0300,0.5900,0.8100
C01213=6.460,-77.460,78.810,0.0400,0.5800,0.8100
C01214=10.550,-78.300,79.670,0.2600,0.3200,0.9100
C01215=12.470,-81.690,81.850,-0.0100,-0.0000,1.0000
C01216=13.580,-87.510,84.880,-0.0700,-0.0100,1.0000
C01217=14.680,-95.270,87.990,-0.1000,-0.0200,0.9900
C01218=15.890,-103.920,90.360,-0.1200,-0.0200,0.9900
C01219=17.370,-111.900,91.520,-0.1200,-0.0400,0.9900
C01220=21.670,-117.740,92.130,-0.0500,-0.0600,1.0000
C01221=28.320,-120.530,92.630,-0.0100,-0.0400,1.0000
C01222=35.970,-119.670,93.130,0.0000,-0.0000,1.0000
C01223=43.870,-117.040,93.460,0.0000,-0.0000,1.0000
C01224=51.740,-113.790,93.460,0.0000,-0.0000,1.0000
C01225=59.190,-110.060,93.130,0.0000,-0.0000,1.0000
C01226=65.200,-105.260,92.630,0.0300,-0.0200,1.0000
C01227=67.930,-98.580,92.130,0.0800,-0.0100,1.0000
C01228=66.840,-91.410,91.520,0.1100,0.0500,0.9900
C01229=62.240,-84.720,90.360,0.1000,0.0700,0.9900
C01230=56.980,-77.740,87.990,0.0900,0.0600,0.9900
C01231=52.280,-71.480,84.880,0.0600,0.0400,1.0000
C01232=48.950,-66.580,81.850,0.0100,0.0000,1.0000
C01233=47.910,-62.820,79.670,-0.4100,0.0500,0.9100
C01234=50.210,-59.340,78.810,-0.4400,0.3800,0.8100
C01235=52.810,-56.920,78.770,-0.4000,0.4400,0.8100
C01236=54.900,-54.900,78.800,-0.4200,0.4200,0.8100
C01237=56.920,-52.810,78.770,-0.4400,0.4000,0.8100
C01238=59.340,-50.210,78.810,-0.3800,0.4400,0.8100
C01239=62.820,-47.910,79.670,-0.0500,0.4100,0.9100
C01240=66.580,-48.950,81.850,-0.0000,-0.0100,1.0000
C01241=71.480,-52.280,84.880,-0.0400,-0.0600,1.0000
C01242=77.740,-56.980,87.990,-0.0600,-0.0900,0.9900
C01243=84.720,-62.240,90.360,-0.0700,-0.1000,0.9900
C01244=91.410,-66.840,91.520,-0.0500,-0.1100,0.9900
C01245=98.580,-67.930,92.130,0.0100,-0.0800,1.0000
C01246=105.260,-65.200,92.630,0.0200,-0.0300,1.0000
C01247=110.060,-59.190,93.130,0.0000,-0.0000,1.0000
C01248=113.790,-51.740,93.460,0.0000,-0.0000,1.0000
C01249=117.040,-43.870,93.460,0.0000,-0.0000,1.0000
C01250=119.670,-35.970,93.130,0.0000,-0.0000,1.0000
C01251=120.530,-28.320,92.630,0.0400,0.0100,1.0000
C01252=117.740,-21.670,92.130,0.0600,0.0500,1.0000
C01253=111.900,-17.370,91.520,0.0400,0.1200,0.9900
C01254=103.920,-15.890,90.360,0.0200,0.1200,0.9900
C01255=95.270,-14.680,87.990,0.0200,0.1000,0.9900
C01256=87.510,-13.580,84.880,0.0100,0.0700,1.0000
C01257=81.690,-12.470,81.850,0.0000,0.0100,1.0000
C01258=78.300,-10.550,79.670,-0.3200,-0.2600,0.9100
C01259=77.460,-6.460,78.810,-0.5800,-0.0400,0.8100
C01260=77.590,-2.910,78.770,-0.5900,0.0300,0.8100
C01261=77.640,0.000,78.800,-0.5900,-0.0000,0.8100
C01262=77.590,2.910,78.770,-0.5900,-0.0300,0.8100
C01263=77.460,6.460,78.810,-0.5800,0.0400,0.8100
C01264=78.300,10.550,79.670,-0.3200,0.2600,0.9100
C01265=81.690,12.470,81.850,0.0000,-0.0100,1.0000
C01266=87.510,13.580,84.880,0.0100,-0.0700,1.0000
C01267=95.270,14.680,87.990,0.0200,-0.1000,0.9900
C01268=103.920,15.890,90.360,0.0200,-0.1200,0.9900
C01269=111.900,17.370,91.520,0.0400,-0.1200,0.9900
C01270=117.740,21.670,92.130,0.0600,-0.0500,1.0000
C01271=120.530,28.320,92.630,0.0400,-0.0100,1.0000
C01272=119.670,35.970,93.130,0.0000,0.0000,1.0000
C01273=117.040,43.870,93.460,0.0000,0.0000,1.0000
C01274=113.790,51.740,93.460,0.0000,0.0000,1.0000
C01275=110.060,59.190,93.130,0.0000,0.0000,1.0000
C01276=105.260,65.200,92.630,0.0200,0.0300,1.0000
C01277=98.580,67.930,92.130,0.0100,0.0800,1.0000
C01278=91.410,66.840,91.520,-0.0500,0.1100,0.9900
C01279=84.720,62.240,90.360,-0.0700,0.1000,0.9900
C01280=77.740,56.980,87.990,-0.0600,0.0900,0.9900
C01281=71.480,52.280,84.880,-0.0400,0.0600,1.0000
C01282=66.580,48.950,81.850,-0.0000,0.0100,1.0000
C01283=62.820,47.910,79.670,-0.0500,-0.4100,0.9100
C01284=59.340,50.210,78.810,-0.3800,-0.4400,0.8100
C01285=56.920,52.810,78.770,-0.4400,-0.4000,0.8100
C01286=54.900,54.900,78.800,-0.4200,-0.4200,0.8100
C01287=52.810,56.920,78.770,-0.4000,-0.4400,0.8100
C01288=50.210,59.340,78.810,-0.4400,-0.3800,0.8100
C01289=47.910,62.820,79.670,-0.4100,-0.0500,0.9100
C01290=48.950,66.580,81.850,0.0100,-0.0000,1.0000
C01291=52.280,71.480,84.880,0.0600,-0.0400,1.0000
C01292=56.980,77.740,87.990,0.0900,-0.0600,0.9900
C01293=62.240,84.720,90.360,0.1000,-0.0700,0.9900
C01294=66.840,91.410,91.520,0.1100,-0.0500,0.9900
C01295=67.930,98.580,92.130,0.0800,0.0100,1.0000
C01296=65.200,105.260,92.630,0.0300,0.0200,1.0000
C01297=59.190,110.060,93.130,0.0000,0.0000,1.0000
C01298=51.740,113.790,93.460,0.0000,0.0000,1.0000
C01299=43.870,117.040,93.460,0.0000,0.0000,1.0000
C01300=35.970,119.670,93.130,0.0000,0.0000,1.0000
C01301=28.320,120.530,92.630,-0.0100,0.0400,1.0000
C01302=21.670,117.740,92.130,-0.0500,0.0600,1.0000
C01303=17.370,111.900,91.520,-0.1200,0.0400,0.9900
C01304=15.890,103.920,90.360,-0.1200,0.0200,0.9900
C01305=14.680,95.270,87.990,-0.1000,0.0200,0.9900
C01306=13.580,87.510,84.880,-0.0700,0.0100,1.0000
C01307=12.470,81.690,81.850,-0.0100,0.0000,1.0000
C01308=10.550,78.300,79.670,0.2600,-0.3200,0.9100
C01309=6.460,77.460,78.810,0.0400,-0.5800,0.8100
C01310=2.910,77.590,78.770,-0.0300,-0.5900,0.8100
C01311=0.000,77.640,78.800,-0.0000,-0.5900,0.8100
C01312=0.000,76.640,80.170,-0.0000,-0.5900,0.8100
C01313=2.820,76.590,80.150,-0.0300,-0.5900,0.8100
C01314=6.300,76.470,80.190,0.0400,-0.5700,0.8200
C01315=10.360,77.350,81.070,0.2500,-0.3100,0.9200
C01316=12.240,80.840,83.310,-0.0100,0.0000,1.0000
C01317=13.330,86.830,86.410,-0.0700,0.0100,1.0000
C01318=14.430,94.770,89.600,-0.1000,0.0200,0.9900
C01319=15.630,103.610,92.010,-0.1200,0.0200,0.9900
C01320=17.100,111.760,93.190,-0.1100,0.0400,0.9900
C01321=21.420,117.710,93.810,-0.0500,0.0600,1.0000
C01322=28.130,120.570,94.320,-0.0100,0.0400,1.0000
C01323=35.850,119.710,94.820,0.0000,0.0000,1.0000
C01324=43.830,117.060,95.160,0.0000,0.0000,1.0000
C01325=51.780,113.770,95.160,0.0000,0.0000,1.0000
C01326=59.300,110.000,94.820,0.0000,0.0000,1.0000
C01327=65.370,105.140,94.320,0.0300,0.0200,1.0000
C01328=68.090,98.380,93.810,0.0800,0.0100,1.0000
C01329=66.930,91.120,93.190,0.1100,-0.0500,0.9900
C01330=62.210,84.320,92.010,0.1000,-0.0700,0.9900
C01331=56.810,77.210,89.600,0.0800,-0.0600,0.9900
C01332=51.970,70.820,86.410,0.0600,-0.0400,1.0000
C01333=48.510,65.820,83.310,0.0100,-0.0100,1.0000
C01334=47.370,62.020,81.070,-0.4000,-0.0400,0.9200
C01335=49.620,58.530,80.190,-0.4400,-0.3800,0.8200
C01336=52.160,56.150,80.150,-0.4000,-0.4300,0.8100
C01337=54.190,54.190,80.170,-0.4100,-0.4100,0.8100
C01338=56.150,52.160,80.150,-0.4300,-0.4000,0.8100
C01339=58.530,49.620,80.190,-0.3800,-0.4400,0.8200
C01340=62.020,47.370,81.070,-0.0400,-0.4000,0.9200
C01341=65.820,48.510,83.310,-0.0100,0.0100,1.0000
C01342=70.820,51.970,86.410,-0.0400,0.0600,1.0000
C01343=77.210,56.810,89.600,-0.0600,0.0800,0.9900
C01344=84.320,62.210,92.010,-0.0700,0.1000,0.9900
C01345=91.120,66.930,93.190,-0.0500,0.1100,0.9900
C01346=98.380,68.090,93.810,0.0100,0.0800,1.0000
C01347=105.140,65.370,94.320,0.0200,0.0300,1.0000
C01348=110.000,59.300,94.820,0.0000,0.0000,1.0000
C01349=113.770,51.780,95.160,0.0000,0.0000,1.0000
C01350=117.060,43.830,95.160,0.0000,0.0000,1.0000
C01351=119.710,35.850,94.820,0.0000,0.0000,1.0000
C01352=120.570,28.130,94.320,0.0400,-0.0100,1.0000
C01353=117.710,21.420,93.810,0.0600,-0.0500,1.0000
C01354=111.760,17.100,93.190,0.0400,-0.1100,0.9900
C01355=103.610,15.630,92.010,0.0200,-0.1200,0.9900
C01356=94.770,14.430,89.600,0.0200,-0.1000,0.9900
C01357=86.830,13.330,86.410,0.0100,-0.0700,1.0000
C01358=80.840,12.240,83.310,0.0000,-0.0100,1.0000
C01359=77.350,10.360,81.070,-0.3100,0.2500,0.9200
C01360=76.470,6.300,80.190,-0.5700,0.0400,0.8200
C01361=76.590,2.820,80.150,-0.5900,-0.0300,0.8100
C01362=76.640,0.000,80.170,-0.5900,-0.0000,0.8100
C01363=76.590,-2.820,80.150,-0.5900,0.0300,0.8100
C01364=76.470,-6.300,80.190,-0.5700,-0.0400,0.8200
C01365=77.350,-10.360,81.070,-0.3100,-0.2500,0.9200
C01366=80.840,-12.240,83.310,0.0000,0.0100,1.0000
C01367=86.830,-13.330,86.410,0.0100,0.0700,1.0000
C01368=94.770,-14.430,89.600,0.0200,0.1000,0.9900
C01369=103.610,-15.630,92.010,0.0200,0.1200,0.9900
C01370=111.760,-17.100,93.190,0.0400,0.1100,0.9900
C01371=117.710,-21.420,93.810,0.0600,0.0500,1.0000
C01372=120.570,-28.130,94.320,0.0400,0.0100,1.0000
C01373=119.710,-35.850,94.820,0.0000,-0.0000,1.0000
C01374=117.060,-43.830,95.160,0.0000,-0.0000,1.0000
C01375=113.770,-51.780,95.160,0.0000,-0.0000,1.0000
C01376=110.000,-59.300,94.820,0.0000,-0.0000,1.0000
C01377=105.140,-65.370,94.320,0.0200,-0.0300,1.0000
C01378=98.380,-68.090,93.810,0.0100,-0.0800,1.0000
C01379=91.120,-66.930,93.190,-0.0500,-0.1100,0.9900
C01380=84.320,-62.210,92.010,-0.0700,-0.1000,0.9900
C01381=77.210,-56.810,89.600,-0.0600,-0.0800,0.9900
C01382=70.820,-51.970,86.410,-0.0400,-0.0600,1.0000
C01383=65.820,-48.510,83.310,-0.0100,-0.0100,1.0000
C01384=62.020,-47.370,81.070,-0.0400,0.4000,0.9200
C01385=58.530,-49.620,80.190,-0.3800,0.4400,0.8200
C01386=56.150,-52.160,80.150,-0.4300,0.4000,0.8100
C01387=54.190,-54.190,80.170,-0.4100,0.4100,0.8100
C01388=52.160,-56.150,80.150,-0.4000,0.4300,0.8100
C01389=49.620,-58.530,80.190,-0.4400,0.3800,0.8200
C01390=47.370,-62.020,81.070,-0.4000,0.0400,0.9200
C01391=48.510,-65.820,83.310,0.0100,0.0100,1.0000
C01392=51.970,-70.820,86.410,0.0600,0.0400,1.0000
C01393=56.810,-77.210,89.600,0.0800,0.0600,0.9900
C01394=62.210,-84.320,92.010,0.1000,0.0700,0.9900
C01395=66.930,-91.120,93.190,0.1100,0.0500,0.9900
C01396=68.090,-98.380,93.810,0.0800,-0.0100,1.0000
C01397=65.370,-105.140,94.320,0.0300,-0.0200,1.0000
C01398=59.300,-110.000,94.820,0.0000,-0.0000,1.0000
C01399=51.780,-113.770,95.160,0.0000,-0.0000,1.0000
C01400=43.830,-117.060,95.160,0.0000,-0.0000,1.0000
C01401=35.850,-119.710,94.820,0.0000,-0.0000,1.0000
C01402=28.130,-120.570,94.320,-0.0100,-0.0400,1.0000
C01403=21.420,-117.710,93.810,-0.0500,-0.0600,1.0000
C01404=17.100,-111.760,93.190,-0.1100,-0.0400,0.9900
C01405=15.630,-103.610,92.010,-0.1200,-0.0200,0.9900
C01406=14.430,-94.770,89.600,-0.1000,-0.0200,0.9900
C01407=13.330,-86.830,86.410,-0.0700,-0.0100,1.0000
C01408=12.240,-80.840,83.310,-0.0100,-0.0000,1.0000
C01409=10.360,-77.350,81.070,0.2500,0.3100,0.9200
C01410=6.300,-76.470,80.190,0.0400,0.5700,0.8200
C01411=2.820,-76.590,80.150,-0.0300,0.5900,0.8100
C01412=0.000,-76.640,80.170,-0.0000,0.5900,0.8100
C01413=0.000,-76.640,80.170,-0.0000,0.5900,0.8100
C01414=-2.820,-76.590,80.150,0.0300,0.5900,0.8100
C01415=-6.300,-76.470,80.190,-0.0400,0.5700,0.8200
C01416=-10.360,-77.350,81.070,-0.2500,0.3100,0.9200
C01417=-12.240,-80.840,83.310,0.0100,-0.0000,1.0000
C01418=-13.330,-86.830,86.410,0.0700,-0.0100,1.0000
C01419=-14.430,-94.770,89.600,0.1000,-0.0200,0.9900
C01420=-15.630,-103.610,92.010,0.1200,-0.0200,0.9900
C01421=-17.100,-111.760,93.190,0.1100,-0.0400,0.9900
C01422=-21.420,-117.710,93.810,0.0500,-0.0600,1.0000
C01423=-28.130,-120.570,94.320,0.0100,-0.0400,1.0000
C01424=-35.850,-119.710,94.820,-0.0000,-0.0000,1.0000
C01425=-43.830,-117.060,95.160,-0.0000,-0.0000,1.0000
C01426=-51.780,-113.770,95.160,-0.0000,-0.0000,1.0000
C01427=-59.300,-110.000,94.820,-0.0000,-0.0000,1.0000
C01428=-65.370,-105.140,94.320,-0.0300,-0.0200,1.0000
C01429=-68.090,-98.380,93.810,-0.0800,-0.0100,1.0000
C01430=-66.930,-91.120,93.190,-0.1100,0.0500,0.9900
C01431=-62.210,-84.320,92.010,-0.1000,0.0700,0.9900
C01432=-56.810,-77.210,89.600,-0.0800,0.0600,0.9900
C01433=-51.970,-70.820,86.410,-0.0600,0.0400,1.0000
C01434=-48.510,-65.820,83.310,-0.0100,0.0100,1.0000
C01435=-47.370,-62.020,81.070,0.4000,0.0400,0.9200
C01436=-49.620,-58.530,80.190,0.4400,0.3800,0.8200
C01437=-52.160,-56.150,80.150,0.4000,0.4300,0.8100
C01438=-54.190,-54.190,80.170,0.4100,0.4100,0.8100
C01439=-56.150,-52.160,80.150,0.4300,0.4000,0.8100
C01440=-58.530,-49.620,80.190,0.3800,0.4400,0.8200
C01441=-62.020,-47.370,81.070,0.0400,0.4000,0.9200
C01442=-65.820,-48.510,83.310,0.0100,-0.0100,1.0000
C01443=-70.820,-51.970,86.410,0.0400,-0.0600,1.0000
C01444=-77.210,-56.810,89.600,0.0600,-0.0800,0.9900
C01445=-84.320,-62.210,92.010,0.0700,-0.1000,0.9900
C01446=-91.120,-66.930,93.190,0.0500,-0.1100,0.9900
C01447=-98.380,-68.090,93.810,-0.0100,-0.0800,1.0000
C01448=-105.140,-65.370,94.320,-0.0200,-0.0300,1.0000
C01449=-110.000,-59.300,94.820,-0.0000,-0.0000,1.0000
C01450=-113.770,-51.780,95.160,-0.0000,-0.0000,1.0000
C01451=-117.060,-43.830,95.160,-0.0000,-0.0000,1.0000
C01452=-119.710,-35.850,94.820,-0.0000,-0.0000,1.0000
C01453=-120.570,-28.130,94.320,-0.0400,0.0100,1.0000
C01454=-117.710,-21.420,93.810,-0.0600,0.0500,1.0000
C01455=-111.760,-17.100,93.190,-0.0400,0.1100,0.9900
C01456=-103.610,-15.630,92.010,-0.0200,0.1200,0.9900
C01457=-94.770,-14.430,89.600,-0.0200,0.1000,0.9900
C01458=-86.830,-13.330,86.410,-0.0100,0.0700,1.0000
C01459=-80.840,-12.240,83.310,-0.0000,0.0100,1.0000
C01460=-77.350,-10.360,81.070,0.3100,-0.2500,0.9200
C01461=-76.470,-6.300,80.190,0.5700,-0.0400,0.8200
C01462=-76.590,-2.820,80.150,0.5900,0.0300,0.8100
C01463=-76.640,0.000,80.170,0.5900,0.0000,0.8100
C01464=-76.590,2.820,80.150,0.5900,-0.0300,0.8100
C01465=-76.470,6.300,80.190,0.5700,0.0400,0.8200
C01466=-77.350,10.360,81.070,0.3100,0.2500,0.9200
C01467=-80.840,12.240,83.310,-0.0000,-0.0100,1.0000
C01468=-86.830,13.330,86.410,-0.0100,-0.0700,1.0000
C01469=-94.770,14.430,89.600,-0.0200,-0.1000,0.9900
C01470=-103.610,15.630,92.010,-0.0200,-0.1200,0.9900
C01471=-111.760,17.100,93.190,-0.0400,-0.1100,0.9900
C01472=-117.710,21.420,93.810,-0.0600,-0.0500,1.0000
C01473=-120.570,28.130,94.320,-0.0400,-0.0100,1.0000
C01474=-119.710,35.850,94.820,-0.0000,0.0000,1.0000
C01475=-117.060,43.830,95.160,-0.0000,0.0000,1.0000
C01476=-113.770,51.780,95.160,-0.0000,0.0000,1.0000
C01477=-110.000,59.300,94.820,-0.0000,0.0000,1.0000
C01478=-105.140,65.370,94.320,-0.0200,0.0300,1.0000
C01479=-98.380,68.090,93.810,-0.0100,0.0800,1.0000
C01480=-91.120,66.930,93.190,0.0500,0.1100,0.9900
C01481=-84.320,62.210,92.010,0.0700,0.1000,0.9900
C01482=-77.210,56.810,89.600,0.0600,0.0800,0.9900
C01483=-70.820,51.970,86.410,0.0400,0.0600,1.0000
C01484=-65.820,48.510,83.310,0.0100,0.0100,1.0000
C01485=-62.020,47.370,81.070,0.0400,-0.4000,0.9200
C01486=-58.530,49.620,80.190,0.3800,-0.4400,0.8200
C01487=-56.150,52.160,80.150,0.4300,-0.4000,0.8100
C01488=-54.190,54.190,80.170,0.4100,-0.4100,0.8100
C01489=-52.160,56.150,80.150,0.4000,-0.4300,0.8100
C01490=-49.620,58.530,80.190,0.4400,-0.3800,0.8200
C01491=-47.370,62.020,81.070,0.4000,-0.0400,0.9200
C01492=-48.510,65.820,83.310,-0.0100,-0.0100,1.0000
C01493=-51.970,70.820,86.410,-0.0600,-0.0400,1.0000
C01494=-56.810,77.210,89.600,-0.0800,-0.0600,0.9900
C01495=-62.210,84.320,92.010,-0.1000,-0.0700,0.9900
C01496=-66.930,91.120,93.190,-0.1100,-0.0500,0.9900
C01497=-68.090,98.380,93.810,-0.0800,0.0100,1.0000
C01498=-65.370,105.140,94.320,-0.0300,0.0200,1.0000
C01499=-59.300,110.000,94.820,-0.0000,0.0000,1.0000
C01500=-51.780,113.770,95.160,-0.0000,0.0000,1.0000
C01501=-43.830,117.060,95.160,-0.0000,0.0000,1.0000
C01502=-35.850,119.710,94.820,-0.0000,0.0000,1.0000
C01503=-28.130,120.570,94.320,0.0100,0.0400,1.0000
C01504=-21.420,117.710,93.810,0.0500,0.0600,1.0000
C01505=-17.100,111.760,93.190,0.1100,0.0400,0.9900
C01506=-15.630,103.610,92.010,0.1200,0.0200,0.9900
C01507=-14.430,94.770,89.600,0.1000,0.0200,0.9900
C01508=-13.330,86.830,86.410,0.0700,0.0100,1.0000
C01509=-12.240,80.840,83.310,0.0100,0.0000,1.0000
C01510=-10.360,77.350,81.070,-0.2500,-0.3100,0.9200
C01511=-6.300,76.470,80.190,-0.0400,-0.5700,0.8200
C01512=-2.820,76.590,80.150,0.0300,-0.5900,0.8100
C01513=0.000,76.640,80.170,-0.0000,-0.5900,0.8100
C01514=0.000,75.650,81.550,-0.0000,-0.5800,0.8200
C01515=-2.730,75.610,81.530,0.0200,-0.5800,0.8200
C01516=-6.150,75.500,81.570,-0.0400,-0.5700,0.8200
C01517=-10.170,76.420,82.480,-0.2500,-0.2900,0.9200
C01518=-12.020,80.010,84.780,0.0200,0.0000,1.0000
C01519=-13.090,86.160,87.960,0.0700,0.0100,1.0000
C01520=-14.180,94.290,91.210,0.1000,0.0200,0.9900
C01521=-15.380,103.310,93.670,0.1100,0.0200,0.9900
C01522=-16.840,111.610,94.870,0.1100,0.0400,0.9900
C01523=-21.180,117.680,95.500,0.0400,0.0600,1.0000
C01524=-27.940,120.600,96.010,0.0100,0.0400,1.0000
C01525=-35.730,119.750,96.520,-0.0000,0.0000,1.0000
C01526=-43.790,117.070,96.850,-0.0000,0.0000,1.0000
C01527=-51.820,113.750,96.850,-0.0000,0.0000,1.0000
C01528=-59.410,109.940,96.520,-0.0000,0.0000,1.0000
C01529=-65.520,105.030,96.010,-0.0300,0.0200,1.0000
C01530=-68.240,98.190,95.500,-0.0700,0.0100,1.0000
C01531=-67.020,90.830,94.870,-0.1000,-0.0500,0.9900
C01532=-62.180,83.930,93.670,-0.0900,-0.0700,0.9900
C01533=-56.650,76.700,91.210,-0.0800,-0.0600,0.9900
C01534=-51.670,70.180,87.960,-0.0600,-0.0400,1.0000
C01535=-48.080,65.080,84.780,-0.0100,-0.0100,1.0000
C01536=-46.840,61.230,82.480,0.3800,-0.0300,0.9200
C01537=-49.040,57.730,81.570,0.4300,-0.3700,0.8200
C01538=-51.530,55.390,81.530,0.3900,-0.4300,0.8200
C01539=-53.490,53.490,81.550,0.4100,-0.4100,0.8200
C01540=-55.390,51.530,81.530,0.4300,-0.3900,0.8200
C01541=-57.730,49.040,81.570,0.3700,-0.4300,0.8200
C01542=-61.230,46.840,82.480,0.0300,-0.3800,0.9200
C01543=-65.080,48.080,84.780,0.0100,0.0100,1.0000
C01544=-70.180,51.670,87.960,0.0400,0.0600,1.0000
C01545=-76.700,56.650,91.210,0.0600,0.0800,0.9900
C01546=-83.930,62.180,93.670,0.0700,0.0900,0.9900
C01547=-90.830,67.020,94.870,0.0500,0.1000,0.9900
C01548=-98.190,68.240,95.500,-0.0100,0.0700,1.0000
C01549=-105.030,65.520,96.010,-0.0200,0.0300,1.0000
C01550=-109.940,59.410,96.520,-0.0000,0.0000,1.0000
C01551=-113.750,51.820,96.850,-0.0000,0.0000,1.0000
C01552=-117.070,43.790,96.850,-0.0000,0.0000,1.0000
C01553=-119.750,35.730,96.520,-0.0000,0.0000,1.0000
C01554=-120.600,27.940,96.010,-0.0400,-0.0100,1.0000
C01555=-117.680,21.180,95.500,-0.0600,-0.0400,1.0000
C01556=-111.610,16.840,94.870,-0.0400,-0.1100,0.9900
C01557=-103.310,15.380,93.670,-0.0200,-0.1100,0.9900
C01558=-94.290,14.180,91.210,-0.0200,-0.1000,0.9900
C01559=-86.160,13.090,87.960,-0.0100,-0.0700,1.0000
C01560=-80.010,12.020,84.780,-0.0000,-0.0200,1.0000
C01561=-76.420,10.170,82.480,0.2900,0.2500,0.9200
C01562=-75.500,6.150,81.570,0.5700,0.0400,0.8200
C01563=-75.610,2.730,81.530,0.5800,-0.0200,0.8200
C01564=-75.650,0.000,81.550,0.5800,0.0000,0.8200
C01565=-75.610,-2.730,81.530,0.5800,0.0200,0.8200
C01566=-75.500,-6.150,81.570,0.5700,-0.0400,0.8200
C01567=-76.420,-10.170,82.480,0.2900,-0.2500,0.9200
C01568=-80.010,-12.020,84.780,-0.0000,0.0200,1.0000
C01569=-86.160,-13.090,87.960,-0.0100,0.0700,1.0000
C01570=-94.290,-14.180,91.210,-0.0200,0.1000,0.9900
C01571=-103.310,-15.380,93.670,-0.0200,0.1100,0.9900
C01572=-111.610,-16.840,94.870,-0.0400,0.1100,0.9900
C01573=-117.680,-21.180,95.500,-0.0600,0.0400,1.0000
C01574=-120.600,-27.940,96.010,-0.0400,0.0100,1.0000
C01575=-119.750,-35.730,96.520,-0.0000,-0.0000,1.0000
C01576=-117.070,-43.790,96.850,-0.0000,-0.0000,1.0000
C01577=-113.750,-51.820,96.850,-0.0000,-0.0000,1.0000
C01578=-109.940,-59.410,96.520,-0.0000,-0.0000,1.0000
C01579=-105.030,-65.520,96.010,-0.0200,-0.0300,1.0000
C01580=-98.190,-68.240,95.500,-0.0100,-0.0700,1.0000
C01581=-90.830,-67.020,94.870,0.0500,-0.1000,0.9900
C01582=-83.930,-62.180,93.670,0.0700,-0.0900,0.9900
C01583=-76.700,-56.650,91.210,0.0600,-0.0800,0.9900
C01584=-70.180,-51.670,87.960,0.0400,-0.0600,1.0000
C01585=-65.080,-48.080,84.780,0.0100,-0.0100,1.0000
C01586=-61.230,-46.840,82.480,0.0300,0.3800,0.9200
C01587=-57.730,-49.040,81.570,0.3700,0.4300,0.8200
C01588=-55.390,-51.530,81.530,0.4300,0.3900,0.8200
C01589=-53.490,-53.490,81.550,0.4100,0.4100,0.8200
C01590=-51.530,-55.390,81.530,0.3900,0.4300,0.8200
C01591=-49.040,-57.730,81.570,0.4300,0.3700,0.8200
C01592=-46.840,-61.230,82.480,0.3800,0.0300,0.9200
C01593=-48.080,-65.080,84.780,-0.0100,0.0100,1.0000
C01594=-51.670,-70.180,87.960,-0.0600,0.0400,1.0000
C01595=-56.650,-76.700,91.210,-0.0800,0.0600,0.9900
C01596=-62.180,-83.930,93.670,-0.0900,0.0700,0.9900
C01597=-67.020,-90.830,94.870,-0.1000,0.0500,0.9900
C01598=-68.240,-98.190,95.500,-0.0700,-0.0100,1.0000
C01599=-65.520,-105.030,96.010,-0.0300,-0.0200,1.0000
C01600=-59.410,-109.940,96.520,-0.0000,-0.0000,1.0000
C01601=-51.820,-113.750,96.850,-0.0000,-0.0000,1.0000
C01602=-43.790,-117.070,96.850,-0.0000,-0.0000,1.0000
C01603=-35.730,-119.750,96.520,-0.0000,-0.0000,1.0000
C01604=-27.940,-120.600,96.010,0.0100,-0.0400,1.0000
C01605=-21.180,-117.680,95.500,0.0400,-0.0600,1.0000
C01606=-16.840,-111.610,94.870,0.1100,-0.0400,0.9900
C01607=-15.380,-103.310,93.670,0.1100,-0.0200,0.9900
C01608=-14.180,-94.290,91.210,0.1000,-0.0200,0.9900
C01609=-13.090,-86.160,87.960,0.0700,-0.0100,1.0000
C01610=-12.020,-80.010,84.780,0.0200,-0.0000,1.0000
C01611=-10.170,-76.420,82.480,-0.2500,0.2900,0.9200
C01612=-6.150,-75.500,81.570,-0.0400,0.5700,0.8200
C01613=-2.730,-75.610,81.530,0.0200,0.5800,0.8200
C01614=0.000,-75.650,81.550,-0.0000,0.5800,0.8200
C01615=0.000,-75.650,81.550,-0.0000,0.5800,0.8200
C01616=2.730,-75.610,81.530,-0.0200,0.5800,0.8200
C01617=6.150,-75.500,81.570,0.0400,0.5700,0.8200
C01618=10.170,-76.420,82.480,0.2500,0.2900,0.9200
C01619=12.020,-80.010,84.780,-0.0200,-0.0000,1.0000
C01620=13.090,-86.160,87.960,-0.0700,-0.0100,1.0000
C01621=14.180,-94.290,91.210,-0.1000,-0.0200,0.9900
C01622=15.380,-103.310,93.670,-0.1100,-0.0200,0.9900
C01623=16.840,-111.610,94.870,-0.1100,-0.0400,0.9900
C01624=21.180,-117.680,95.500,-0.0400,-0.0600,1.0000
C01625=27.940,-120.600,96.010,-0.0100,-0.0400,1.0000
C01626=35.730,-119.750,96.520,0.0000,-0.0000,1.0000
C01627=43.790,-117.070,96.850,0.0000,-0.0000,1.0000
C01628=51.820,-113.750,96.850,0.0000,-0.0000,1.0000
C01629=59.410,-109.940,96.520,0.0000,-0.0000,1.0000
C01630=65.520,-105.030,96.010,0.0300,-0.0200,1.0000
C01631=68.240,-98.190,95.500,0.0700,-0.0100,1.0000
C01632=67.020,-90.830,94.870,0.1000,0.0500,0.9900
C01633=62.180,-83.930,93.670,0.0900,0.0700,0.9900
C01634=56.650,-76.700,91.210,0.0800,0.0600,0.9900
C01635=51.670,-70.180,87.960,0.0600,0.0400,1.0000
C01636=48.080,-65.080,84.780,0.0100,0.0100,1.0000
C01637=46.840,-61.230,82.480,-0.3800,0.0300,0.9200
C01638=49.040,-57.730,81.570,-0.4300,0.3700,0.8200
C01639=51.530,-55.390,81.530,-0.3900,0.4300,0.8200
C01640=53.490,-53.490,81.550,-0.4100,0.4100,0.8200
C01641=55.390,-51.530,81.530,-0.4300,0.3900,0.8200
C01642=57.730,-49.040,81.570,-0.3700,0.4300,0.8200
C01643=61.230,-46.840,82.480,-0.0300,0.3800,0.9200
C01644=65.080,-48.080,84.780,-0.0100,-0.0100,1.0000
C01645=70.180,-51.670,87.960,-0.0400,-0.0600,1.0000
C01646=76.700,-56.650,91.210,-0.0600,-0.0800,0.9900
C01647=83.930,-62.180,93.670,-0.0700,-0.0900,0.9900
C01648=90.830,-67.020,94.870,-0.0500,-0.1000,0.9900
C01649=98.190,-68.240,95.500,0.0100,-0.0700,1.0000
C01650=105.030,-65.520,96.010,0.0200,-0.0300,1.0000
C01651=109.940,-59.410,96.520,0.0000,-0.0000,1.0000
C01652=113.750,-51.820,96.850,0.0000,-0.0000,1.0000
C01653=117.070,-43.790,96.850,0.0000,-0.0000,1.0000
C01654=119.750,-35.730,96.520,0.0000,-0.0000,1.0000
C01655=120.600,-27.940,96.010,0.0400,0.0100,1.0000
C01656=117.680,-21.180,95.500,0.0600,0.0400,1.0000
C01657=111.610,-16.840,94.870,0.0400,0.1100,0.9900
C01658=103.310,-15.380,93.670,0.0200,0.1100,0.9900
C01659=94.290,-14.180,91.210,0.0200,0.1000,0.9900
C01660=86.160,-13.090,87.960,0.0100,0.0700,1.0000
C01661=80.010,-12.020,84.780,0.0000,0.0200,1.0000
C01662=76.420,-10.170,82.480,-0.2900,-0.2500,0.9200
C01663=75.500,-6.150,81.570,-0.5700,-0.0400,0.8200
C01664=75.610,-2.730,81.530,-0.5800,0.0200,0.8200
C01665=75.650,0.000,81.550,-0.5800,-0.0000,0.8200
C01666=75.610,2.730,81.530,-0.5800,-0.0200,0.8200
C01667=75.500,6.150,81.570,-0.5700,0.0400,0.8200
C01668=76.420,10.170,82.480,-0.2900,0.2500,0.9200
C01669=80.010,12.020,84.780,0.0000,-0.0200,1.0000
C01670=86.160,13.090,87.960,0.0100,-0.0700,1.0000
C01671=94.290,14.180,91.210,0.0200,-0.1000,0.9900
C01672=103.310,15.380,93.670,0.0200,-0.1100,0.9900
C01673=111.610,16.840,94.870,0.0400,-0.1100,0.9900
C01674=117.680,21.180,95.500,0.0600,-0.0400,1.0000
C01675=120.600,27.940,96.010,0.0400,-0.0100,1.0000
C01676=119.750,35.730,96.520,0.0000,0.0000,1.0000
C01677=117.070,43.790,96.850,0.0000,0.0000,1.0000
C01678=113.750,51.820,96.850,0.0000,0.0000,1.0000
C01679=109.940,59.410,96.520,0.0000,0.0000,1.0000
C01680=105.030,65.520,96.010,0.0200,0.0300,1.0000
C01681=98.190,68.240,95.500,0.0100,0.0700,1.0000
C01682=90.830,67.020,94.870,-0.0500,0.1000,0.9900
C01683=83.930,62.180,93.670,-0.0700,0.0900,0.9900
C01684=76.700,56.650,91.210,-0.0600,0.0800,0.9900
C01685=70.180,51.670,87.960,-0.0400,0.0600,1.0000
C01686=65.080,48.080,84.780,-0.0100,0.0100,1.0000
C01687=61.230,46.840,82.480,-0.0300,-0.3800,0.9200
C01688=57.730,49.040,81.570,-0.3700,-0.4300,0.8200
C01689=55.390,51.530,81.530,-0.4300,-0.3900,0.8200
C01690=53.490,53.490,81.550,-0.4100,-0.4100,0.8200
C01691=51.530,55.390,81.530,-0.3900,-0.4300,0.8200
C01692=49.040,57.730,81.570,-0.4300,-0.3700,0.8200
C01693=46.840,61.230,82.480,-0.3800,-0.0300,0.9200
C01694=48.080,65.080,84.780,0.0100,-0.0100,1.0000
C01695=51.670,70.180,87.960,0.0600,-0.0400,1.0000
C01696=56.650,76.700,91.210,0.0800,-0.0600,0.9900
C01697=62.180,83.930,93.670,0.0900,-0.0700,0.9900
C01698=67.020,90.830,94.870,0.1000,-0.0500,0.9900
C01699=68.240,98.190,95.500,0.0700,0.0100,1.0000
C01700=65.520,105.030,96.010,0.0300,0.0200,1.0000
C01701=59.410,109.940,96.520,0.0000,0.0000,1.0000
C01702=51.820,113.750,96.850,0.0000,0.0000,1.0000
C01703=43.790,117.070,96.850,0.0000,0.0000,1.0000
C01704=35.730,119.750,96.520,0.0000,0.0000,1.0000
C01705=27.940,120.600,96.010,-0.0100,0.0400,1.0000
C01706=21.180,117.680,95.500,-0.0400,0.0600,1.0000
C01707=16.840,111.610,94.870,-0.1100,0.0400,0.9900
C01708=15.380,103.310,93.670,-0.1100,0.0200,0.9900
C01709=14.180,94.290,91.210,-0.1000,0.0200,0.9900
C01710=13.090,86.160,87.960,-0.0700,0.0100,1.0000
C01711=12.020,80.010,84.780,-0.0200,0.0000,1.0000
C01712=10.170,76.420,82.480,0.2500,-0.2900,0.9200
C01713=6.150,75.500,81.570,0.0400,-0.5700,0.8200
C01714=2.730,75.610,81.530,-0.0200,-0.5800,0.8200
C01715=0.000,75.650,81.550,-0.0000,-0.5800,0.8200
C01716=0.000,74.670,82.950,-0.0000,-0.5700,0.8200
C01717=2.640,74.630,82.920,-0.0200,-0.5700,0.8200
C01718=6.000,74.530,82.960,0.0500,-0.5600,0.8300
C01719=9.990,75.490,83.900,0.2500,-0.2800,0.9300
C01720=11.810,79.200,86.260,-0.0200,0.0000,1.0000
C01721=12.850,85.500,89.510,-0.0700,0.0100,1.0000
C01722=13.940,93.820,92.830,-0.1000,0.0200,1.0000
C01723=15.150,103.030,95.330,-0.1100,0.0200,0.9900
C01724=16.590,111.480,96.540,-0.1000,0.0400,0.9900
C01725=20.950,117.650,97.180,-0.0400,0.0500,1.0000
C01726=27.760,120.640,97.700,-0.0100,0.0300,1.0000
C01727=35.620,119.790,98.210,0.0000,0.0000,1.0000
C01728=43.760,117.090,98.550,0.0000,0.0000,1.0000
C01729=51.850,113.730,98.550,0.0000,0.0000,1.0000
C01730=59.520,109.890,98.210,0.0000,0.0000,1.0000
C01731=65.670,104.930,97.700,0.0300,0.0200,1.0000
C01732=68.380,98.010,97.180,0.0700,0.0100,1.0000
C01733=67.100,90.560,96.540,0.1000,-0.0500,0.9900
C01734=62.140,83.560,95.330,0.0900,-0.0700,0.9900
C01735=56.490,76.200,92.830,0.0800,-0.0600,1.0000
C01736=51.370,69.550,89.510,0.0600,-0.0400,1.0000
C01737=47.650,64.350,86.260,0.0200,-0.0100,1.0000
C01738=46.320,60.450,83.900,-0.3700,-0.0200,0.9300
C01739=48.460,56.950,82.960,-0.4300,-0.3600,0.8300
C01740=50.910,54.640,82.920,-0.3900,-0.4200,0.8200
C01741=52.800,52.800,82.950,-0.4000,-0.4000,0.8200
C01742=54.640,50.910,82.920,-0.4200,-0.3900,0.8200
C01743=56.950,48.460,82.960,-0.3600,-0.4300,0.8300
C01744=60.450,46.320,83.900,-0.0200,-0.3700,0.9300
C01745=64.350,47.650,86.260,-0.0100,0.0200,1.0000
C01746=69.550,51.370,89.510,-0.0400,0.0600,1.0000
C01747=76.200,56.490,92.830,-0.0600,0.0800,1.0000
C01748=83.560,62.140,95.330,-0.0700,0.0900,0.9900
C01749=90.560,67.100,96.540,-0.0500,0.1000,0.9900
C01750=98.010,68.380,97.180,0.0100,0.0700,1.0000
C01751=104.930,65.670,97.700,0.0200,0.0300,1.0000
C01752=109.890,59.520,98.210,0.0000,0.0000,1.0000
C01753=113.730,51.850,98.550,0.0000,0.0000,1.0000
C01754=117.090,43.760,98.550,0.0000,0.0000,1.0000
C01755=119.790,35.620,98.210,0.0000,0.0000,1.0000
C01756=120.640,27.760,97.700,0.0300,-0.0100,1.0000
C01757=117.650,20.950,97.180,0.0500,-0.0400,1.0000
C01758=111.480,16.590,96.540,0.0400,-0.1000,0.9900
C01759=103.030,15.150,95.330,0.0200,-0.1100,0.9900
C01760=93.820,13.940,92.830,0.0200,-0.1000,1.0000
C01761=85.500,12.850,89.510,0.0100,-0.0700,1.0000
C01762=79.200,11.810,86.260,0.0000,-0.0200,1.0000
C01763=75.490,9.990,83.900,-0.2800,0.2500,0.9300
C01764=74.530,6.000,82.960,-0.5600,0.0500,0.8300
C01765=74.630,2.640,82.920,-0.5700,-0.0200,0.8200
C01766=74.670,0.000,82.950,-0.5700,-0.0000,0.8200
C01767=74.630,-2.640,82.920,-0.5700,0.0200,0.8200
C01768=74.530,-6.000,82.960,-0.5600,-0.0500,0.8300
C01769=75.490,-9.990,83.900,-0.2800,-0.2500,0.9300
C01770=79.200,-11.810,86.260,0.0000,0.0200,1.0000
C01771=85.500,-12.850,89.510,0.0100,0.0700,1.0000
C01772=93.820,-13.940,92.830,0.0200,0.1000,1.0000
C01773=103.030,-15.150,95.330,0.0200,0.1100,0.9900
C01774=111.480,-16.590,96.540,0.0400,0.1000,0.9900
C01775=117.650,-20.950,97.180,0.0500,0.0400,1.0000
C01776=120.640,-27.760,97.700,0.0300,0.0100,1.0000
C01777=119.790,-35.620,98.210,0.0000,-0.0000,1.0000
C01778=117.090,-43.760,98.550,0.0000,-0.0000,1.0000
C01779=113.730,-51.850,98.550,0.0000,-0.0000,1.0000
C01780=109.890,-59.520,98.210,0.0000,-0.0000,1.0000
C01781=104.930,-65.670,97.700,0.0200,-0.0300,1.0000
C01782=98.010,-68.380,97.180,0.0100,-0.0700,1.0000
C01783=90.560,-67.100,96.540,-0.0500,-0.1000,0.9900
C01784=83.560,-62.140,95.330,-0.0700,-0.0900,0.9900
C01785=76.200,-56.490,92.830,-0.0600,-0.0800,1.0000
C01786=69.550,-51.370,89.510,-0.0400,-0.0600,1.0000
C01787=64.350,-47.650,86.260,-0.0100,-0.0200,1.0000
C01788=60.450,-46.320,83.900,-0.0200,0.3700,0.9300
C01789=56.950,-48.460,82.960,-0.3600,0.4300,0.8300
C01790=54.640,-50.910,82.920,-0.4200,0.3900,0.8200
C01791=52.800,-52.800,82.950,-0.4000,0.4000,0.8200
C01792=50.910,-54.640,82.920,-0.3900,0.4200,0.8200
C01793=48.460,-56.950,82.960,-0.4300,0.3600,0.8300
C01794=46.320,-60.450,83.900,-0.3700,0.0200,0.9300
C01795=47.650,-64.350,86.260,0.0200,0.0100,1.0000
C01796=51.370,-69.550,89.510,0.0600,0.0400,1.0000
C01797=56.490,-76.200,92.830,0.0800,0.0600,1.0000
C01798=62.140,-83.560,95.330,0.0900,0.0700,0.9900
C01799=67.100,-90.560,96.540,0.1000,0.0500,0.9900
C01800=68.380,-98.010,97.180,0.0700,-0.0100,1.0000
C01801=65.670,-104.930,97.700,0.0300,-0.0200,1.0000
C01802=59.520,-109.890,98.210,0.0000,-0.0000,1.0000
C01803=51.850,-113.730,98.550,0.0000,-0.0000,1.0000
C01804=43.760,-117.090,98.550,0.0000,-0.0000,1.0000
C01805=35.620,-119.790,98.210,0.0000,-0.0000,1.0000
C01806=27.760,-120.640,97.700,-0.0100,-0.0300,1.0000
C01807=20.950,-117.650,97.180,-0.0400,-0.0500,1.0000
C01808=16.590,-111.480,96.540,-0.1000,-0.0400,0.9900
C01809=15.150,-103.030,95.330,-0.1100,-0.0200,0.9900
C01810=13.940,-93.820,92.830,-0.1000,-0.0200,1.0000
C01811=12.850,-85.500,89.510,-0.0700,-0.0100,1.0000
C01812=11.810,-79.200,86.260,-0.0200,-0.0000,1.0000
C01813=9.990,-75.490,83.900,0.2500,0.2800,0.9300
C01814=6.000,-74.530,82.960,0.0500,0.5600,0.8300
C01815=2.640,-74.630,82.920,-0.0200,0.5700,0.8200
C01816=0.000,-74.670,82.950,-0.0000,0.5700,0.8200
C01817=0.000,-74.670,82.950,-0.0000,0.5700,0.8200
C01818=-2.640,-74.630,82.920,0.0200,0.5700,0.8200
C01819=-6.000,-74.530,82.960,-0.0500,0.5600,0.8300
C01820=-9.990,-75.490,83.900,-0.2500,0.2800,0.9300
C01821=-11.810,-79.200,86.260,0.0200,-0.0000,1.0000
C01822=-12.850,-85.500,89.510,0.0700,-0.0100,1.0000
C01823=-13.940,-93.820,92.830,0.1000,-0.0200,1.0000
C01824=-15.150,-103.030,95.330,0.1100,-0.0200,0.9900
C01825=-16.590,-111.480,96.540,0.1000,-0.0400,0.9900
C01826=-20.950,-117.650,97.180,0.0400,-0.0500,1.0000
C01827=-27.760,-120.640,97.700,0.0100,-0.0300,1.0000
C01828=-35.620,-119.790,98.210,-0.0000,-0.0000,1.0000
C01829=-43.760,-117.090,98.550,-0.0000,-0.0000,1.0000
C01830=-51.850,-113.730,98.550,-0.0000,-0.0000,1.0000
C01831=-59.520,-109.890,98.210,-0.0000,-0.0000,1.0000
C01832=-65.670,-104.930,97.700,-0.0300,-0.0200,1.0000
C01833=-68.380,-98.010,97.180,-0.0700,-0.0100,1.0000
C01834=-67.100,-90.560,96.540,-0.1000,0.0500,0.9900
C01835=-62.140,-83.560,95.330,-0.0900,0.0700,0.9900
C01836=-56.490,-76.200,92.830,-0.0800,0.0600,1.0000
C01837=-51.370,-69.550,89.510,-0.0600,0.0400,1.0000
C01838=-47.650,-64.350,86.260,-0.0200,0.0100,1.0000
C01839=-46.320,-60.450,83.900,0.3700,0.0200,0.9300
C01840=-48.460,-56.950,82.960,0.4300,0.3600,0.8300
C01841=-50.910,-54.640,82.920,0.3900,0.4200,0.8200
C01842=-52.800,-52.800,82.950,0.4000,0.4000,0.8200
C01843=-54.640,-50.910,82.920,0.4200,0.3900,0.8200
C01844=-56.950,-48.460,82.960,0.3600,0.4300,0.8300
C01845=-60.450,-46.320,83.900,0.0200,0.3700,0.9300
C01846=-64.350,-47.650,86.260,0.0100,-0.0200,1.0000
C01847=-69.550,-51.370,89.510,0.0400,-0.0600,1.0000
C01848=-76.200,-56.490,92.830,0.0600,-0.0800,1.0000
C01849=-83.560,-62.140,95.330,0.0700,-0.0900,0.9900
C01850=-90.560,-67.100,96.540,0.0500,-0.1000,0.9900
C01851=-98.010,-68.380,97.180,-0.0100,-0.0700,1.0000
C01852=-104.930,-65.670,97.700,-0.0200,-0.0300,1.0000
C01853=-109.890,-59.520,98.210,-0.0000,-0.0000,1.0000
C01854=-113.730,-51.850,98.550,-0.0000,-0.0000,1.0000
C01855=-117.090,-43.760,98.550,-0.0000,-0.0000,1.0000
C01856=-119.790,-35.620,98.210,-0.0000,-0.0000,1.0000
C01857=-120.640,-27.760,97.700,-0.0300,0.0100,1.0000
C01858=-117.650,-20.950,97.180,-0.0500,0.0400,1.0000
C01859=-111.480,-16.590,96.540,-0.0400,0.1000,0.9900
C01860=-103.030,-15.150,95.330,-0.0200,0.1100,0.9900
C01861=-93.820,-13.940,92.830,-0.0200,0.1000,1.0000
C01862=-85.500,-12.850,89.510,-0.0100,0.0700,1.0000
C01863=-79.200,-11.810,86.260,-0.0000,0.0200,1.0000
C01864=-75.490,-9.990,83.900,0.2800,-0.2500,0.9300
C01865=-74.530,-6.000,82.960,0.5600,-0.0500,0.8300
C01866=-74.630,-2.640,82.920,0.5700,0.0200,0.8200
C01867=-74.670,0.000,82.950,0.5700,0.0000,0.8200
C01868=-74.630,2.640,82.920,0.5700,-0.0200,0.8200
C01869=-74.530,6.000,82.960,0.5600,0.0500,0.8300
C01870=-75.490,9.990,83.900,0.2800,0.2500,0.9300
C01871=-79.200,11.810,86.260,-0.0000,-0.0200,1.0000
C01872=-85.500,12.850,89.510,-0.0100,-0.0700,1.0000
C01873=-93.820,13.940,92.830,-0.0200,-0.1000,1.0000
C01874=-103.030,15.150,95.330,-0.0200,-0.1100,0.9900
C01875=-111.480,16.590,96.540,-0.0400,-0.1000,0.9900
C01876=-117.650,20.950,97.180,-0.0500,-0.0400,1.0000
C01877=-120.640,27.760,97.700,-0.0300,-0.0100,1.0000
C01878=-119.790,35.620,98.210,-0.0000,0.0000,1.0000
C01879=-117.090,43.760,98.550,-0.0000,0.0000,1.0000
C01880=-113.730,51.850,98.550,-0.0000,0.0000,1.0000
C01881=-109.890,59.520,98.210,-0.0000,0.0000,1.0000
C01882=-104.930,65.670,97.700,-0.0200,0.0300,1.0000
C01883=-98.010,68.380,97.180,-0.0100,0.0700,1.0000
C01884=-90.560,67.100,96.540,0.0500,0.1000,0.9900
C01885=-83.560,62.140,95.330,0.0700,0.0900,0.9900
C01886=-76.200,56.490,92.830,0.0600,0.0800,1.0000
C01887=-69.550,51.370,89.510,0.0400,0.0600,1.0000
C01888=-64.350,47.650,86.260,0.0100,0.0200,1.0000
C01889=-60.450,46.320,83.900,0.0200,-0.3700,0.9300
C01890=-56.950,48.460,82.960,0.3600,-0.4300,0.8300
C01891=-54.640,50.910,82.920,0.4200,-0.3900,0.8200
C01892=-52.800,52.800,82.950,0.4000,-0.4000,0.8200
C01893=-50.910,54.640,82.920,0.3900,-0.4200,0.8200
C01894=-48.460,56.950,82.960,0.4300,-0.3600,0.8300
C01895=-46.320,60.450,83.900,0.3700,-0.0200,0.9300
C01896=-47.650,64.350,86.260,-0.0200,-0.0100,1.0000
C01897=-51.370,69.550,89.510,-0.0600,-0.0400,1.0000
C01898=-56.490,76.200,92.830,-0.0800,-0.0600,1.0000
C01899=-62.140,83.560,95.330,-0.0900,-0.0700,0.9900
C01900=-67.100,90.560,96.540,-0.1000,-0.0500,0.9900
C01901=-68.380,98.010,97.180,-0.0700,0.0100,1.0000
C01902=-65.670,104.930,97.700,-0.0300,0.0200,1.0000
C01903=-59.520,109.890,98.210,-0.0000,0.0000,1.0000
C01904=-51.850,113.730,98.550,-0.0000,0.0000,1.0000
C01905=-43.760,117.090,98.550,-0.0000,0.0000,1.0000
C01906=-35.620,119.790,98.210,-0.0000,0.0000,1.0000
C01907=-27.760,120.640,97.700,0.0100,0.0300,1.0000
C01908=-20.950,117.650,97.180,0.0400,0.0500,1.0000
C01909=-16.590,111.480,96.540,0.1000,0.0400,0.9900
C01910=-15.150,103.030,95.330,0.1100,0.0200,0.9900
C01911=-13.940,93.820,92.830,0.1000,0.0200,1.0000
C01912=-12.850,85.500,89.510,0.0700,0.0100,1.0000
C01913=-11.810,79.200,86.260,0.0200,0.0000,1.0000
C01914=-9.990,75.490,83.900,-0.2500,-0.2800,0.9300
C01915=-6.000,74.530,82.960,-0.0500,-0.5600,0.8300
C01916=-2.640,74.630,82.920,0.0200,-0.5700,0.8200
C01917=0.000,74.670,82.950,-0.0000,-0.5700,0.8200
C01918=0.000,73.710,84.350,-0.0000,-0.5600,0.8300
C01919=-2.550,73.670,84.320,0.0200,-0.5600,0.8300
C01920=-5.850,73.580,84.360,-0.0500,-0.5500,0.8400
C01921=-9.810,74.590,85.320,-0.2400,-0.2600,0.9300
C01922=-11.600,78.400,87.740,0.0300,0.0100,1.0000
C01923=-12.630,84.870,91.070,0.0700,0.0100,1.0000
C01924=-13.710,93.380,94.450,0.0900,0.0100,1.0000
C01925=-14.920,102.760,96.990,0.1000,0.0200,0.9900
C01926=-16.350,111.350,98.220,0.1000,0.0300,0.9900
C01927=-20.730,117.630,98.870,0.0400,0.0500,1.0000
C01928=-27.590,120.670,99.390,0.0000,0.0300,1.0000
C01929=-35.520,119.820,99.910,-0.0000,0.0000,1.0000
C01930=-43.720,117.100,100.250,-0.0000,0.0000,1.0000
C01931=-51.890,113.720,100.250,-0.0000,0.0000,1.0000
C01932=-59.610,109.840,99.910,-0.0000,0.0000,1.0000
C01933=-65.820,104.830,99.390,-0.0300,0.0200,1.0000
C01934=-68.520,97.840,98.870,-0.0700,0.0100,1.0000
C01935=-67.170,90.300,98.220,-0.0900,-0.0500,0.9900
C01936=-62.110,83.210,96.990,-0.0900,-0.0600,0.9900
C01937=-56.330,75.720,94.450,-0.0800,-0.0600,1.0000
C01938=-51.080,68.940,91.070,-0.0600,-0.0400,1.0000
C01939=-47.240,63.640,87.740,-0.0200,-0.0100,1.0000
C01940=-45.800,59.680,85.320,0.3600,-0.0200,0.9300
C01941=-47.890,56.170,84.360,0.4200,-0.3500,0.8400
C01942=-50.290,53.900,84.320,0.3800,-0.4100,0.8300
C01943=-52.120,52.120,84.350,0.4000,-0.4000,0.8300
C01944=-53.900,50.290,84.320,0.4100,-0.3800,0.8300
